	// EtherCAT device
	stText_EC_OpState_Error					: ST_Text := (
												wsNameId:= "EC_OpState_Error",
												wsName:= "EC-Error(OpState)");
	stText_EC_DeviceState_Init				: ST_Text := (
												wsNameId:= "EC_DeviceState_Init",
												wsName:= "EtherCAT Device State: INIT");
	stText_EC_DeviceState_Preop				: ST_Text := (
												wsNameId:= "EC_DeviceState_Preop",
												wsName:= "EtherCAT Device State: Pre-Operational");
	stText_EC_DeviceState_Bootstrap			: ST_Text := (
												wsNameId:= "EC_DeviceState_Bootstrap",
												wsName:= "EtherCAT Device State: Bootstrap");
	stText_EC_DeviceState_Safeop			: ST_Text := (
												wsNameId:= "EC_DeviceState_Safeop",
												wsName:= "EtherCAT Device State: Safe-Operational");
	stText_EC_DeviceState_Op				: ST_Text := (
												wsNameId:= "EC_DeviceState_Op",
												wsName:= "EtherCAT Device State: Operational");
	stText_EC_DeviceState_Error				: ST_Text := (
												wsNameId:= "EC_DeviceState_Error",
												wsName:= "EtherCAT Device State: Error");
	stText_EC_DeviceState_InvalidVprs		: ST_Text := (
												wsNameId:= "EC_DeviceState_InvalidVprs",
												wsName:= "EtherCAT Device State: Invalid VendorID, Productcode, revisionnumber or serialnumber");
	stText_EC_DeviceState_InitCmdError		: ST_Text := (
												wsNameId:= "EC_DeviceState_InitCmdError",
												wsName:= "EtherCAT Device State: INIT command error");
	stText_EC_DeviceState_Undefined			: ST_Text := (
												wsNameId:= "EC_DeviceState_Undefined",
												wsName:= "EtherCAT Device State: Undefined");
												
	// EtherCAT link state
	stText_EC_LinkState_Ok					: ST_Text := (
												wsNameId:= "EC_LinkState_Ok",
												wsName:= "EtherCAT Link State: OK");
	stText_EC_LinkState_NotPresent			: ST_Text := (
												wsNameId:= "EC_LinkState_NotPresent",
												wsName:= "EtherCAT Link State: no EtherCAT communication with slave");
	stText_EC_LinkState_WithoutCom			: ST_Text := (
												wsNameId:= "EC_LinkState_WithoutCom",
												wsName:= "EtherCAT Link State: error on port X. Port has a link, but no communication");
	stText_EC_LinkState_MissingLink			: ST_Text := (
												wsNameId:= "EC_LinkState_MissingLink",
												wsName:= "EtherCAT Link State: Missing link on port X");
	stText_EC_LinkState_AdditionalLink		: ST_Text := (
												wsNameId:= "EC_LinkState_AdditionalLink",
												wsName:= "EtherCAT Link State: Additional link on port X");
	stText_EC_LinkState_PortA				: ST_Text := (
												wsNameId:= "EC_LinkState_PortA",
												wsName:= "EtherCAT Link State: Error communication port A");
	stText_EC_LinkState_PortB				: ST_Text := (
												wsNameId:= "EC_LinkState_PortB",
												wsName:= "EtherCAT Link State: Error communication port B");
	stText_EC_LinkState_PortC				: ST_Text := (
												wsNameId:= "EC_LinkState_PortC",
												wsName:= "EtherCAT Link State: Error communication port C");
	stText_EC_LinkState_PortD				: ST_Text := (
												wsNameId:= "EC_LinkState_PortD",
												wsName:= "EtherCAT Link State: Error communication port D");
	stText_EC_LinkState_Undefined			: ST_Text := (
												wsNameId:= "EC_LinkState_Undefined",
												wsName:= "EtherCAT Link State: Undefined");

	// ProfiNet device
	stText_PN_Device_Error					: ST_Text := (
												wsNameId:= "PN_Device_Error",
												wsName:= "ProfiNet Device Status");

	// IO-Link device
	stText_IOL_Device_Error					: ST_Text := (
												wsNameId:= "IOL_Device_Error",
												wsName:= "IO-Link Device Status");
												
END_STRUCT
END_TYPE

// ---- POUs/HMI/_Structures/_Common/ST_DefaultHmiToPlc.TcDUT
TYPE ST_DefaultHmiToPlc :
STRUCT
	// default HMI items	
	bStart			: BOOL;
	bStop, bFastStop: BOOL;
	bReset			: BOOL;
	bStep			: BOOL;
	bHome			: BOOL;
	
	bOpModeManual	: BOOL;
	bOpModeAuto		: BOOL;
	bOpModeStep		: BOOL;
	
	eSafetyOpMode	: E_Opmode;
END_STRUCT
END_TYPE

// ---- POUs/Items/TcaCarrier/Enumerations/eTcaCarrierCmd.TcDUT
{attribute 'qualified_only'}
{attribute 'strict'}
{attribute 'to_string'}
TYPE eTcaCarrierCmd :
(
	noCmd := 0,
	emptyPlaces,
	fillPlaces,
	RestorePlaces,
	ConfigCarrier
);
END_TYPE

// ---- POUs/Items/TcaCarrier/Enumerations/eTcaCarrierLayout.TcDUT
{attribute 'qualified_only'}
TYPE eTcaCarrierLayout :
(
	undefined := 0,
	Layout1,
	Layout2,
	Layout3,
	Layout4,
	Layout5,
	Bulk
);
END_TYPE

// ---- POUs/Items/TcaCarrier/Structures/TcaCarrierConfig.TcDUT
TYPE TcaCarrierConfig :
STRUCT	
	/// Geometry
	Layout : eTcaCarrierLayout;		
	Dimension : ST_Coordinate;
	
	PositionsInRow : INT;			// Numbers of Positions in first Row
	RowDistance : REAL;		// Distance from one Row to the other
	PositionsInColumn : INT;			// Numbers of Positions in one Column
	ColumnDistance : REAL;		// Distance from one Column to the other
	CoordinateFirstWorkpiece : ST_Coordinate;
		
	InitialStatus : eTcaWorkpieceStatus;
	RequestStatus : eTcaWorkpieceStatus;	
	
END_STRUCT
END_TYPE

// ---- POUs/Items/TcaCarrier/Structures/TcaCarrierData.TcDUT
TYPE TcaCarrierData :
STRUCT	
	Enabled : BOOL;
	Id : INT;
	//Source		: E_Station;
	//Logging : WSTRING;	// Information in csv, xml or json Format
	Error : BOOL;	

	WorkpiecesEnabled : ARRAY[0..TcaCarrier.MAX_WORKPIECEPLACES] OF BOOL;
	WorkpiecesData : ARRAY[0..TcaCarrier.MAX_WORKPIECEPLACES] OF TcaWorkpieceData;		

END_STRUCT
END_TYPE

// ---- POUs/Items/TcaCarrier/Structures/TcaCarrierService.TcDUT
TYPE TcaCarrierService :
STRUCT

END_STRUCT
END_TYPE

// ---- POUs/Items/TcaTrolley/Structures/TcaTrolleyConfig.TcDUT
TYPE TcaTrolleyConfig : 
STRUCT	
	/// Geometry
	NumberOfCarriers : INT := 40;
	RackOrigin : ST_Coordinate;
	RackDivision : LREAL;
	CarrierDistance : LREAL;
	
	//InitialStatus : eTcaWorkpieceStatus;
	//RequestStatus : eTcaWorkpieceStatus;	
	
	CarrierConfig : TcaCarrierConfig;
	
END_STRUCT
END_TYPE

// ---- POUs/Items/TcaTrolley/Structures/TcaTrolleyData.TcDUT
TYPE TcaTrolleyData : 
STRUCT
	Exist : BOOL;
	Id : INT;
	//Logging : WSTRING;	// Information in csv, xml or json Format
	Error : BOOL;
	
	CarriersEnabled : ARRAY[0..TcaCarrier.MAX_WORKPIECEPLACES] OF BOOL;
	CarriersData : ARRAY[0..TcaTrolley.MAX_CARRIERPLACES] OF TcaCarrierData;
	
END_STRUCT
END_TYPE

// ---- POUs/Items/TcaTrolley/Structures/TcaTrolleyService.TcDUT
TYPE TcaTrolleyService :
STRUCT
	DisableCarriers		: BOOL;
	EnableCarriers		: BOOL;
	FillWithEmptyCarriers : BOOL;
	FillWithFinishedCarriers : BOOL;
	FillWithInitialCarriers : BOOL;
END_STRUCT
END_TYPE

// ---- POUs/Items/TcaWorkpiece/Enumerations/eTcaWorkpieceShape.TcDUT
{attribute 'qualified_only'}
{attribute 'strict'}
{attribute 'to_string'}
TYPE eTcaWorkpieceShape :
(
	undefined := 0,
	roll,
	ring,
	plate,
	other,
	
	MAXSIZE
);
END_TYPE

// ---- POUs/Items/TcaWorkpiece/Enumerations/eTcaWorkpieceStatus.TcDUT
{attribute 'qualified_only'}
{attribute 'to_string'}
TYPE eTcaWorkpieceStatus :
(
	undefined := 0, //leer
	noProcessDone, // grau
	laserProcessDone, // blau
	bondingAgentProcessDone, // orange
	castingProcessDone, //  violett
	finishProcessDone, //grün
	

	MAXSIZE
);
END_TYPE

// ---- POUs/Items/TcaWorkpiece/Structures/TcaWorkpieceData.TcDUT
TYPE TcaWorkpieceData : 
STRUCT
	Id : INT;	// <> 0 Workpiece Present 
	Error : BOOL;
	Exist : BOOL;
	SerialNumber : STRING;
	CurrentStatus : eTcaWorkpieceStatus;
	InitialStatus : eTcaWorkpieceStatus;
	RequestStatus : eTcaWorkpieceStatus;
	//Shape : eTcaWorkpieceShape;
	//Dimension : ST_Coordinate;
	TimeStampChanged : DT;
	Logging : WSTRING;	// Information in csv, xml or json Format
	
END_STRUCT
END_TYPE

// ---- POUs/Plant/_Enumerations/E_Module.TcDUT
//{attribute 'qualified_only'}
//{attribute 'strict'}
TYPE E_Module :
(
	eModule_none := 0,
	eModule_M001,
		
	/// has to be set to last index for array bounds!
	eModule_nMaxIdx
);
END_TYPE

// ---- POUs/Plant/_Enumerations/E_PlantSettings.TcDUT
//{attribute 'qualified_only'}
//{attribute 'strict'}
{attribute 'to_string'}
{attribute 'to_wstring'}
TYPE E_PlantSettings :
(
	//ePlant_Settings_none := 0,
	ePlantSetting_RecipeName,		// Name of the recipe
	ePlantSetting_RecipeComment,	// Comment
	ePlantSetting_PlantName,		// Plant name
	ePlantSetting_PlantNumber,		// Plant number
	
	//ePlantSetting_OvenHgPickUpDepthZ,	// Einfahrtiefe HG - Oven Z-Achse
	//
	//ePlantSetting_StorageHgSafetyDistZ,	// Sicherheitsabstand HG - Storage Z-Achse
	//
	//ePlantSetting_StorageOffsetUpY,	// HG-Offset oberhalb der Storage-Palette in Y-Richtung [mm]
	//ePlantSetting_StorageOffsetDnY, // HG-Offset unterhalb der Storage-Palette in Y-Richtung [mm]
	
	/// has to be set to last index for array bounds!
	ePlantSetting_nMaxIdx	
);
END_TYPE

// ---- POUs/Plant/_Enumerations/E_ProductionSettings.TcDUT
//{attribute 'qualified_only'}
//{attribute 'strict'}
{attribute 'to_string'}
{attribute 'to_wstring'}
TYPE E_ProductionSettings :
(
	//eProduction_Settings_none := 0,
	eProductionSettings_Override,		// override
	eProductionSettings_OrderNumber,	// order

	/// has to be set to last index for array bounds!
	eProductionSettings_nMaxIdx	
);
END_TYPE

// ---- POUs/Plant/_Enumerations/E_ProductSettings.TcDUT
//{attribute 'qualified_only'}
//{attribute 'strict'}
{attribute 'to_string'}
{attribute 'to_wstring'}
TYPE E_ProductSettings :
(
	//eProduct_Settings_none := 0,
	eProductSettings_ProductNumber,	// product nb.
	eProductSettings_ProductName,	// product name
	eProductSettings_ProductType, 	// product type
	
	//eProductSettings_Speed,			// speed [m/min]
	
	//eProductSettings_TrolleyDevisionX,	// Teilung des Trolley-Racks in X-Richtung [mm]
	//eProductSettings_TrolleyFirstPosY, 	// Erte Position im Trolley-Racks in Y-Richtung [mm]
	//eProductSettings_TrolleyCountY, 	// Letzte Position im Trolley-Racks in Y-Richtung [mm]
	//eProductSettings_TrolleyDevisionY,	// Teilung des Trolley-Racks in Y-Richtung [mm]
	//eProductSettings_TrolleyOffsetUpY,	// HG-Offset oberhalb der Trolley-Palette in Y-Richtung [mm]
	//eProductSettings_TrolleyOffsetDnY,	// HG-Offset unterhalb der Trolley-Palette in Y-Richtung [mm]
	
	eProductSettings_TrolleyNumberOfCarriers,
	eProductSettings_TrolleyRackOriginX,
	eProductSettings_TrolleyRackOriginY,
	eProductSettings_TrolleyRackOriginZ,
	eProductSettings_TrolleyRackDivision,
	eProductSettings_TrolleyCarrierDistance,
	
	eProductSettings_CarrierLayout,	
	eProductSettings_CarrierDimensionX,
	eProductSettings_CarrierDimensionY,
	eProductSettings_CarrierPositionsInRow,			// Numbers of Positions in first Row
	eProductSettings_CarrierRowDistance,		// Distance from one Row to the other
	eProductSettings_CarrierPositionsInColumn,			// Numbers of Positions in one Column
	eProductSettings_CarrierColumnDistance,		// Distance from one Column to the other
	eProductSettings_CarrierCoordinateFirstWorkpieceX,
	eProductSettings_CarrierCoordinateFirstWorkpieceY,
	eProductSettings_CarrierInitialStatus,
	eProductSettings_CarrierRequestStatus,	
	
	
	eProductSettings_HeatingPlateEnable,
	eProductSettings_HeatingPlateTemperatur,	
	
	/// has to be set to last index for array bounds!
	eProductSettings_nMaxIdx	
);
END_TYPE

// ---- POUs/Plant/_Enumerations/E_Station.TcDUT
//{attribute 'qualified_only'}
//{attribute 'strict'}
TYPE E_Station :
(
	eStation_none := 0,
	eStation_ST010_OvenA := 1,
	eStation_ST020_OvenB := 2,
	eStation_ST030_Handling := 3,
	eStation_ST040_Storage := 4,
	eStation_ST050_Mould := 5,
	
	/// has to be set to last index for array bounds!
	eStation_nMaxIdx
);
END_TYPE

// ---- POUs/Plant/M001_Module/_Enumerations/E_M001_Settings.TcDUT
//{attribute 'qualified_only'}
//{attribute 'strict'}
{attribute 'to_string'}
{attribute 'to_wstring'}
TYPE E_M001_Settings :
(
	//eSt001_Settings_none := 0,
	
	eM001_Settings_Deaktiv,		// Station deaktivieren
	eM001_Settings_Autohome,	// automatic home with start button
	
	//eM001_Settings_PalletLayout,	// Palettenlayout (1-4)
	
	/// has to be set to last index for array bounds!
	eM001_Settings_nMaxIdx	
);
END_TYPE

// ---- POUs/Plant/M001_Module/_Structures/ST_M001_HMI_IN.TcDUT
TYPE ST_M001_HMI_IN :
STRUCT
	bQuit : BOOL;
	//bJogVm : BOOL;
END_STRUCT
END_TYPE

// ---- POUs/Plant/M001_Module/_Structures/ST_M001_Interface.TcDUT
TYPE ST_M001_Interface :
STRUCT
	bRunCycle,
	bEmptyPlant : BOOL;
END_STRUCT
END_TYPE

// ---- POUs/Plant/M001_Module/_Structures/ST_M001_HMI_OUT.TcDUT
TYPE ST_M001_HMI_OUT :
STRUCT
	//fSpeed : LREAL;
END_STRUCT
END_TYPE

// ---- POUs/Plant/M001_Module/_Structures/ST_M001_IO.TcDUT
TYPE ST_M001_IO :
STRUCT
	stIn 	AT%I* : ST_M001_IO_IN;
	stOut 	AT%Q* : ST_M001_IO_OUT;
END_STRUCT
END_TYPE

// ---- POUs/Plant/M001_Module/_Structures/ST_M001_IO_IN.TcDUT
TYPE ST_M001_IO_IN :
STRUCT	
	// inputs	
	//bPwrCircBreakerOk	: BOOL;
END_STRUCT
END_TYPE

// ---- POUs/Plant/M001_Module/_Structures/ST_M001_IO_OUT.TcDUT
TYPE ST_M001_IO_OUT :
STRUCT
END_STRUCT
END_TYPE

// ---- POUs/Plant/ST010_OvenA/_Structures/ST_St010_HMI_IN.TcDUT
TYPE ST_St010_HMI_IN :
STRUCT
	bJogUp : BOOL; // Tippen Vor; DT-WH, 2FDI-NO; P10A-52SJ1
	bJogDown : BOOL; // Tippen Zurück; DT-BK, 2FDI-NO; P10A-52SJ3
	
	bJogCh1Ouside : BOOL;
	bJogCh1Inside : BOOL;
	
	bJogCh2Ouside : BOOL;
	bJogCh2Inside : BOOL;
	
	bManual : BOOL;
	bQuit : BOOL;
	
	bJog : BOOL;
	bSpeed : BOOL;
	
END_STRUCT
END_TYPE

// ---- POUs/Plant/ST010_OvenA/_Structures/ST_St010_Interface.TcDUT
TYPE ST_St010_Interface :
STRUCT
	bEnableSequence,	// enable to main module
	
	bResponseChkIndex,
	bResponseIsEmptySlot,
	bResponseOpn	: BOOL;	// handshake response segment open
	iConfirmPosition	: INT;	// handshake confirm segment open @ x,y index
	
	Trolley			: TcaTrolley;
END_STRUCT
END_TYPE

// ---- POUs/Plant/ST010_OvenA/_Structures/ST_St010_HMI_IN_OUT.TcDUT
TYPE ST_St010_HMI_IN_OUT : //EXTENDS ST_HMI_TR_CMD :
STRUCT
END_STRUCT
END_TYPE

// ---- POUs/Plant/ST020_OvenB/_Enumerations/E_St020_Settings.TcDUT
//{attribute 'qualified_only'}
//{attribute 'strict'}
{attribute 'to_string'}
{attribute 'to_wstring'}
TYPE E_St020_Settings :
(
	//eSt020_Settings_none := 0,
	
	eSt020_Settings_Station_Deaktiv,	// Station deaktivieren
	eSt020_Settings_Autohome,			// automatic home with start button
	
	eSt020_Settings_HomeSpeed,			// Homing-Geschwindigkeit [mm/s]
	eSt020_Settings_JogSpeed,			// Tippgeschwindigkeit [mm/s]
	eSt020_Settings_WorkSpeed,			// Automatik-Geschwindigkeit [mm/s]
	eSt020_Settings_JogSpeedCh,			// Tippgeschwindigkeit CH-Achsen [mm/s]
	eSt020_Settings_WorkSpeedCh,		// Automatik-Geschwindigkeit CH-Achsen [mm/s]

	eSt020_Settings_AxisRefPos,			// Referenzposition Achse [mm]
	eSt020_Settings_PosHome,			// Homeposition [mm]
	eSt020_Settings_PosWork,			// Mitnehmerposition unteres Segment [mm]
	
	eSt020_Settings_PosHomeCh,			// Homeposition CH-Achsen [mm]
	eSt020_Settings_PosWorkCh,			// Arbeitsposition CH-Achsen [mm]
	
	eSt020_Settings_OvenFixPartHeight,	// Festteilhöhe [mm]
	eSt020_Settings_OvenSegmentHeight,	// Festteilhöhe [mm]
	
	eSt020_Settings_OvenMiddlePointX,	// Mittelpunnkt in X-Richtung [mm]
	eSt020_Settings_OvenOffsetY,		// Y-Offset Ofen [mm]
	eSt020_Settings_OvenPickUpDepthZ,	// Teach-Position, Storage 2 Z [mm]
	
	eSt020_Settings_XPosRp1,			// Teach-Position, Ofen B, RP 1 X [mm]
	eSt020_Settings_YPosRp1,			// Teach-Position, Ofen B, RP 1 Y [mm]
	eSt020_Settings_ZPosRp1,			// Teach-Position, Ofen B, RP 1 Z [mm]
	                                                           
	eSt020_Settings_XPosRp2,			// Teach-Position, Ofen B, RP 2 X [mm]
	eSt020_Settings_YPosRp2,			// Teach-Position, Ofen B, RP 2 Y [mm]
	eSt020_Settings_ZPosRp2,			// Teach-Position, Ofen B, RP 2 Z [mm]
	
	/// has to be set to last index for array bounds!
	eSt020_Settings_nMaxIdx	
);
END_TYPE

// ---- POUs/Plant/ST020_OvenB/_Structures/ST_St020_HMI_IN_OUT.TcDUT
TYPE ST_St020_HMI_IN_OUT : // EXTENDS ST_HMI_TR_CMD :
STRUCT
END_STRUCT
END_TYPE

// ---- POUs/Plant/ST020_OvenB/_Structures/ST_St020_HMI_IN.TcDUT
TYPE ST_St020_HMI_IN :
STRUCT	
	bJogUp : BOOL; // Tippen Vor; DT-WH, 2FDI-NO; P10A-52SJ1
	bJogDown : BOOL; // Tippen Zurück; DT-BK, 2FDI-NO; P10A-52SJ3
	
	bJogCh1Ouside : BOOL;
	bJogCh1Inside : BOOL;
	
	bJogCh2Ouside : BOOL;
	bJogCh2Inside : BOOL;
	
	bManual : BOOL;
	bQuit : BOOL;
	
	bJog : BOOL;
	bSpeed : BOOL;
END_STRUCT
END_TYPE

// ---- POUs/Plant/ST020_OvenB/_Structures/ST_St020_Interface.TcDUT
TYPE ST_St020_Interface :
STRUCT
	bEnableSequence,	// enable to main module
	
	bResponseChkIndex,
	bResponseIsEmptySlot,
	bResponseOpn	: BOOL;	// handshake response segment open
	iConfirmPosition	: INT;	// handshake confirm segment open @ x,y index
	
	Trolley			: TcaTrolley;
END_STRUCT
END_TYPE

// ---- POUs/Plant/ST020_OvenB/_Structures/ST_St020_IO.TcDUT
TYPE ST_St020_IO :
STRUCT
	stIn	AT%I* : ST_St020_IO_IN;
	stOut	AT%Q* : ST_St020_IO_OUT;
	stHeatingPlateIO : ST_FurnaceIO;
END_STRUCT
END_TYPE

// ---- POUs/Plant/ST020_OvenB/_Structures/ST_St020_IO_IN.TcDUT
TYPE ST_St020_IO_IN :
STRUCT	
	// inputs
	bRefpos	: BOOL;	// Sensor | Oven | Referenzposition | BMK: =P260+xyz- | Terminal: .: | Tc3Hmi
END_STRUCT
END_TYPE

// ---- POUs/Plant/ST020_OvenB/_Structures/ST_St020_IO_OUT.TcDUT
TYPE ST_St020_IO_OUT :
STRUCT
	bOvenFan :BOOL;
END_STRUCT
END_TYPE

// ---- POUs/Plant/ST020_OvenB/_Structures/ST_St020_HMI_OUT.TcDUT
TYPE ST_St020_HMI_OUT :
STRUCT
	//Trolley	: ST_Trolley;
END_STRUCT
END_TYPE

// ---- POUs/Plant/ST030_Handling/_Enumerations/E_St030_Command.TcDUT
{attribute 'qualified_only'}
{attribute 'strict'}
{attribute 'to_string'}
TYPE E_St030_Command :
(
	eSt030_Command_none := 0,
	eSt030_Command_OvenA_Get,
	eSt030_Command_OvenA_Put,
	
	eSt030_Command_OvenB_Get,
	eSt030_Command_OvenB_Put,
	
	eSt030_Command_Storage_Get,
	eSt030_Command_Storage_Put
);
END_TYPE

// ---- POUs/Plant/ST030_Handling/_Enumerations/E_St030_EmptySlotChk.TcDUT
{attribute 'qualified_only'}
{attribute 'strict'}
{attribute 'to_string'}
TYPE E_St030_EmptySlotChk :
(
	eSt030_EmptySlotChk_none := 0,
	eSt030_EmptySlotChk_Empty,
	eSt030_EmptySlotChk_NotEmpty
);
END_TYPE

// ---- POUs/Plant/ST030_Handling/_Enumerations/E_St030_Settings.TcDUT
//{attribute 'qualified_only'}
//{attribute 'strict'}
{attribute 'to_string'}
{attribute 'to_wstring'}
TYPE E_St030_Settings :
(
	//eSt030_Settings_none := 0,
	
	eSt030_Settings_Station_Deaktiv,	// Station deaktivieren
	eSt030_Settings_Autohome,			// automatic home with start button
	
	eSt030_Settings_XHomeSpeed,			// Homing-Geschwindigkeit X [mm/s]
	eSt030_Settings_XJogSpeed,			// Tippgeschwindigkeit X [mm/s]
	eSt030_Settings_XWorkSpeed,			// Automatik-Geschwindigkeit X [mm/s]
	
	eSt030_Settings_YHomeSpeed,			// Homing-Geschwindigkeit Y [mm/s]
	eSt030_Settings_YJogSpeed,			// Tippgeschwindigkeit Y [mm/s]
	eSt030_Settings_YWorkSpeed,			// Automatik-Geschwindigkeit Y [mm/s]
	
	eSt030_Settings_ZHomeSpeed,			// Homing-Geschwindigkeit Z [mm/s]
	eSt030_Settings_ZJogSpeed,			// Tippgeschwindigkeit Z [mm/s]
	eSt030_Settings_ZWorkSpeed,			// Automatik-Geschwindigkeit Z [mm/s]
	
	eSt030_Settings_AxisRefPosX,		// reference pos axis HG X
	eSt030_Settings_AxisRefPosY,		// reference pos axis HG Y
	eSt030_Settings_AxisRefPosZ,		// reference pos axis HG Z
	
	eSt030_Settings_XPosHome,			// Homeposition X [mm]
	eSt030_Settings_YPosHome,			// Homeposition Y [mm]
	eSt030_Settings_ZPosHome,			// Homeposition Z [mm]

	
	eSt030_Settings_XPosOv2Rp1,			// Teach-Position, Ofen 2, RP 1 X [mm]
	eSt030_Settings_YPosOv2Rp1,			// Teach-Position, Ofen 2, RP 1 Y [mm]
	eSt030_Settings_ZPosOv2Rp1,			// Teach-Position, Ofen 2, RP 1 Z [mm]

	eSt030_Settings_XPosOv2Rp2,			// Teach-Position, Ofen 2, RP 2 X [mm]
	eSt030_Settings_YPosOv2Rp2,			// Teach-Position, Ofen 2, RP 2 Y [mm]
	eSt030_Settings_ZPosOv2Rp2,			// Teach-Position, Ofen 2, RP 2 Z [mm]
	
	
	/// has to be set to last index for array bounds!
	eSt030_Settings_nMaxIdx
);
END_TYPE

// ---- POUs/Plant/ST030_Handling/_Structures/ST_St030_HMI_OUT.TcDUT
TYPE ST_St030_HMI_OUT :
STRUCT
	//Pallet	: ST_Pallet;
END_STRUCT
END_TYPE

// ---- POUs/Plant/ST030_Handling/_Structures/ST_St030_HMI_IN.TcDUT
TYPE ST_St030_HMI_IN :
STRUCT
	bJogXP		: BOOL; // Tippen Vor; DT-WH, 2FDI-NO; P10A-52SJ1
	bJogXN		: BOOL; // Tippen Zurück; DT-BK, 2FDI-NO; P10A-52SJ3
	
	bJogYP		: BOOL; // Tippen Vor; DT-WH, 2FDI-NO; P10A-52SJ1
	bJogYN		: BOOL; // Tippen Zurück; DT-BK, 2FDI-NO; P10A-52SJ3
	
	bJogZP		: BOOL; 
	bJogZN		: BOOL; 
	
	bManual : BOOL;
	bQuit :  BOOL;
		
	bJog : BOOL;
	bSpeed : BOOL;
END_STRUCT
END_TYPE

// ---- POUs/Plant/ST030_Handling/_Structures/ST_St030_Interface.TcDUT
TYPE ST_St030_Interface :
STRUCT
	bEnable,
	bEnableOvenAxis,

	bReqestOvenA,			// request entry to stations
	bReqestOvenA_ChkIndex,
	bReqestOvenB,
	bReqestOvenB_ChkIndex,
	bReqestStorage,
	bReqestStorage_ChkIndex	: BOOL;	
	
	// current pallet on GH
	Pallet			: TcaCarrier;
	Source			: E_Station;
	
	// active / requested HG command
	CommandRequest	: ST_St030_Command;
	ActiveCommand	: ST_St030_Command;
END_STRUCT
END_TYPE

// ---- POUs/Plant/ST030_Handling/_Structures/ST_St030_Command.TcDUT
TYPE ST_St030_Command :
STRUCT
	Command : E_St030_Command;
	Position : INT;
	//IndexX,
	//IndexY	: INT;
END_STRUCT
END_TYPE

// ---- POUs/Plant/ST030_Handling/_Structures/ST_St030_IO.TcDUT
TYPE ST_St030_IO :
STRUCT
	stIn	AT%I* : ST_St030_IO_IN;
	stOut	AT%Q* : ST_St030_IO_OUT;
END_STRUCT
END_TYPE

// ---- POUs/Plant/ST030_Handling/_Structures/ST_St030_IO_IN.TcDUT
TYPE ST_St030_IO_IN :
STRUCT
	// inputs handling
	bRefposX	: BOOL;	// Sensor | Handling | Referenzposition X | BMK: =P260+xyz- | Terminal: .: | Tc3Hmi
	bRefposY	: BOOL;	// Sensor | Handling | Referenzposition Y | BMK: =P260+xyz- | Terminal: .: | Tc3Hmi
	bRefposZ	: BOOL;	// Sensor | Handling | Referenzposition Z | BMK: =P260+xyz- | Terminal: .: | Tc3Hmi
	
	fMeasurementA : DINT;	// Sensor | Handling | S1 | BMK: =P260+xyz- | Terminal: .: | Tc3Hmi
	fMeasurementB : DINT;	// Sensor | Handling | S2 | BMK: =P260+xyz- | Terminal: .: | Tc3Hmi
END_STRUCT
END_TYPE

// ---- POUs/Plant/ST030_Handling/_Structures/ST_St030_IO_OUT.TcDUT
TYPE ST_St030_IO_OUT :
STRUCT
	// outputs handling
END_STRUCT
END_TYPE

// ---- POUs/Plant/ST030_Handling/_Structures/ST_St030_HMI_IN_OUT.TcDUT
TYPE ST_St030_HMI_IN_OUT ://EXTENDS ST_HMI_PL_CMD :
STRUCT
END_STRUCT
END_TYPE

// ---- POUs/Plant/ST030_Handling/_Structures/ST_XZ_Point.TcDUT
TYPE ST_XZ_Point :
STRUCT
	X,
	Z : LREAL;
END_STRUCT
END_TYPE

// ---- POUs/Plant/ST040_Storage/_Enumerations/E_St040_Settings.TcDUT
//{attribute 'qualified_only'}
//{attribute 'strict'}
{attribute 'to_string'}
{attribute 'to_wstring'}
TYPE E_St040_Settings :
(
	//eSt040_Settings_none := 0,
	
	eSt040_Settings_Station_Deaktiv,	// Station deaktivieren
	eSt040_Settings_Autohome,			// automatic home with start button
	
	eSt040_Settings_JogSpeed,			// Tippgeschwindigkeit [mm/s]
	eSt040_Settings_WorkSpeed,			// Automatik-Geschwindigkeit  [mm/s]
	
	eSt040_Settings_PosHome,			// Homeposition [mm]
	eSt040_Settings_PosWork,			// Arbeitsposition [mm]
	
	eSt040_Settings_XPosStor1,			// Teach-Position, Storage 1 X [mm]
	eSt040_Settings_YPosStor1,			// Teach-Position, Storage 1 Y [mm]
	eSt040_Settings_ZPosStor1,			// Teach-Position, Storage 1 Z [mm]
	    
	eSt040_Settings_XPosStor2,			// Teach-Position, Storage 2 X [mm]
	eSt040_Settings_YPosStor2,			// Teach-Position, Storage 2 Y [mm]
	eSt040_Settings_ZPosStor2,			// Teach-Position, Storage 2 Z [mm]
	
	
	/// has to be set to last index for array bounds!
	eSt040_Settings_nMaxIdx	
);
END_TYPE

// ---- POUs/Plant/ST040_Storage/_Structures/ST_St040_HMI_IN.TcDUT
TYPE ST_St040_HMI_IN :
STRUCT
	bJog01Up		: BOOL; // Tippen Vor; DT-WH, 2FDI-NO; P10A-52SJ1
	bJog01Down		: BOOL; // Tippen Zurück; DT-BK, 2FDI-NO; P10A-52SJ3
	
	bJog02Up	 	: BOOL; 
	bJog02Down	: BOOL; 	
	
	bManual : BOOL;
	bQuit :  BOOL;
	
	bJog : BOOL;
	bSpeed : BOOL;

END_STRUCT
END_TYPE

// ---- POUs/Plant/ST040_Storage/_Structures/ST_St040_HMI_IN_OUT.TcDUT
TYPE ST_St040_HMI_IN_OUT : //EXTENDS ST_HMI_PL_CMD :
STRUCT
	// pallet index on storage
	Idx		: INT;
END_STRUCT
END_TYPE

// ---- POUs/Plant/ST040_Storage/_Structures/ST_St040_HMI_OUT.TcDUT
TYPE ST_St040_HMI_OUT :
STRUCT
	//Pallet1,
	//Pallet2	: ST_Pallet;
END_STRUCT
END_TYPE

// ---- POUs/Plant/ST040_Storage/_Structures/ST_St040_IO.TcDUT
TYPE ST_St040_IO :
STRUCT
	stIn	AT%I* : ST_St040_IO_IN;
	stOut	AT%Q* : ST_St040_IO_OUT;
END_STRUCT
END_TYPE

// ---- POUs/Plant/ST040_Storage/_Structures/ST_St040_IO_IN.TcDUT
TYPE ST_St040_IO_IN :
STRUCT
END_STRUCT
END_TYPE

// ---- POUs/Plant/ST040_Storage/_Structures/ST_St040_IO_OUT.TcDUT
TYPE ST_St040_IO_OUT :
STRUCT
	// outputs OptischeKontrolle	
	nCamPrgAs	: INT;
	nCamPrgBs	: INT;
	
	bLedAs		: BOOL;
	bLedBs		: BOOL;
END_STRUCT
END_TYPE

// ---- POUs/Plant/ST040_Storage/_Structures/ST_St040_Interface.TcDUT
TYPE ST_St040_Interface :
STRUCT
	bEnable,				// enable to main module
	
	bResponseChkIndex,
	bResponseEmptyAtIndex,
	bResponseOpn	: BOOL;	// handshake response open
	iConfirmPosition 	: INT;	// handshake confirm open @ index
	
	Pallet1,
	Pallet2	: TcaCarrier;
	
	Source1,	
	Source2			: E_Station;
END_STRUCT
END_TYPE

// ---- POUs/Plant/ST050_Mould/_Enumerations/E_St050_Settings.TcDUT
//{attribute 'qualified_only'}
//{attribute 'strict'}
{attribute 'to_string'}
{attribute 'to_wstring'}
TYPE E_St050_Settings :
(
	//eSt050_Settings_none := 0,
	
	eSt050_Settings_Station_Deaktiv,	// Station deaktivieren
	eSt050_Settings_Autohome,			// automatic home with start button

	
	/// has to be set to last index for array bounds!
	eSt050_Settings_nMaxIdx	
);
END_TYPE

// ---- POUs/Plant/ST050_Mould/_Structures/ST_St050_Interface.TcDUT
TYPE ST_St050_Interface :
STRUCT
	bEnableHG	: BOOL; // enable handling
	
	bReqS1Empty,
	bReqS2Empty,
	bReqS1Unfinished,
	bReqS2Unfinished,
	bReqS1NoCarrier,
	bReqS2NoCarrier	: BOOL;
END_STRUCT
END_TYPE

// ---- POUs/Plant/ST050_Mould/_Structures/ST_St050_IO.TcDUT
TYPE ST_St050_IO :
STRUCT
	stIn	AT%I* : ST_St050_IO_IN;
	stOut	AT%Q* : ST_St050_IO_OUT;
END_STRUCT
END_TYPE

// ---- POUs/Plant/ST050_Mould/_Structures/ST_St050_IO_IN.TcDUT
TYPE ST_St050_IO_IN :
STRUCT
	aFromEngelRaw	: ARRAY[0..41] OF BYTE;
	bRequestOpenProtectionDoor : BOOL;
END_STRUCT
END_TYPE

// ---- POUs/Plant/ST050_Mould/_Structures/ST_St050_IO_OUT.TcDUT
TYPE ST_St050_IO_OUT :
STRUCT
	aToEngelRaw	: ARRAY[0..41] OF BYTE;
	bReleaseSafetyGate : BOOL;
END_STRUCT
END_TYPE

// ---- POUs/Plant/ST050_Mould/_Structures/TcaEngelCastingCarrierInput.TcDUT
TYPE TcaEngelCastingCarrierInput : // ENGEL SPS -> ASMA SPS
STRUCT
	LifeCounter : UINT;
	
	
	// Modus bzw Status der Gießmaschine und Roboter
	AutoMode : BOOL;		// Roboter und Gießmaschine im zyklischen Automatikbetrieb
	SemiAutoMode : BOOL;	// Roboter und Gießmaschine im sequentiellen Halb-Automatikbetrieb
	ManualMode : BOOL;		// Roboter und Gießmaschine befinden sich in Handbetrieb
	Error : BOOL;			// Roboter bzw. Gießmaschine hat Error
	ErrorID : UINT;			// ErrorID
	
	// Überwachung und Kontrolle der Roboterposition
	Moving : BOOL;				// Roboter in Bewegung
	ParkPosition : BOOL;		// Roboter in Wartepostion
	OutsideStorage_1 : BOOL;	// Roboter außerhalb Ablage 1
	OutsideStorage_2 : BOOL;	// Roboter außerhalb Ablage 2

	// Allgemeine Sicherheit                    	
	SafetyAreaSafe : BOOL;	// Schutztüren geschlossen & quittiert		

	// Anforderung eines Werkstückträgers
	// Wird ein leerer Werkstückablageplatz oder ein Einleigeteil benötigt muss für den jeweiligen Ablageplatz
	// ein Job angefrgt werden.
	// Wenn kein Werkstückträger benötigt wird, kann auch dieser Job erteilt werden (z.B. bei Produktionsende)
	
	JobForStorage_1 : TcaEngelCastingCarrierJob;	// Anforderung eines Werkstückträgers für Ablage 1
	JobForStorage_2 : TcaEngelCastingCarrierJob;	// Anforderung eines Werkstückträgers für Ablage 2
	
	// Status des Werkstückträgers
	// Beim Entnehmen und Bestücken eines Werkstückes durch den Engel Roboter wird die Statusstruktur aktualisiert
	
	Storage_1 : TcaEngelCastingCarrierStatus;	// aktueller Status des Werkstückträgers in Ablage 1
	Storage_2 : TcaEngelCastingCarrierStatus;	// aktueller Status des Werkstückträgers in Ablage 2
	
END_STRUCT
END_TYPE

// ---- POUs/Plant/ST050_Mould/_Structures/TcaEngelCastingCarrierJob.TcDUT
TYPE TcaEngelCastingCarrierJob :
STRUCT
	RequestNoCarrier : BOOL;	// TRUE wenn kein neuer Werkstückträger benötigt wird -> Ablage wird leer gemacht
	RequestCarrier : BOOL;		// TRUE wenn ein neuer Werkstückträger benötigt wird
	CarrierId : INT;			// ID vom Werkstückträger, Geometrischen Daten werden auf der Engel Steuerung verwaltet
	Empty : BOOL;				// TRUE wenn ein Werkstückträger mir leeren Plätzen benötigt wird
	Unfinished : BOOL;			// TRUE wenn ein Werkstückträger mit unfertigen Werkstücken benötigt wird
END_STRUCT
END_TYPE

// ---- POUs/Plant/ST050_Mould/_Structures/TcaEngelCastingCarrierJobStatus.TcDUT
TYPE TcaEngelCastingCarrierJobStatus :
STRUCT
	CarrierPresent : BOOL;						// TRUE wenn ein Werkstückträger abgelegt wurde
	Carrier : TcaEngelCastingCarrierStatus;		// Status des Carriers der abgelegt wurde
	Done : BOOL;								// Job wurde erfolgreich ausgeführt
	Busy : BOOL;								// Job wird ausgeführt
	Error : BOOL;								// Job endet mit Fehler
	ErrorID : UINT;								// TODO: Welche unterschiedlichen Fehler sollen berücksichtigt werden? z.b: kein Blech, Ofentür offen, Wagen ist zum wechseln, ...								
END_STRUCT
END_TYPE

// ---- POUs/Plant/ST050_Mould/_Structures/TcaEngelCastingCarrierOutput.TcDUT
TYPE TcaEngelCastingCarrierOutput :	// ASMA SPS -> ENGEL SPS
STRUCT
	LifeCounter : UINT;
	
	// Status der Peripherie
	Ready : BOOL;			// Bereit zum Entgegennehmen von Jobs
	Busy : BOOL;			// Peripherie ist in Arbeit/ Bewegung
	Error : BOOL;			// Peripherie hat Error
	ErrorID : INT;			// ErrorID
	
	// Überwachung und Kontrolle der Ablageposition und des Handlings
	PermitRoboterHandling : BOOL; 	// Bewegungen des Engel Roboters erlauben (freie Fahrt im gesamten Bewgungsbereich)(
	PermitStorage_1 : BOOL;			// Zugriff auf Ablage 1 erlauben (aufnehmen und ablegen)
	PermitStorage_2 : BOOL;			// Zugriff auf Ablage 1 erlauben (aufnehmen und ablegen)
	                    	
	// Allgemeine Sicherheit						
	SafetyAreaRequest : BOOL; 	// Anforderung Schutztüre
	SafetyDoorRelease : BOOL;	// freigabe zum öffnen der Schutztüre
	
	// Status der Jobs
	JobStatusForStorage_1 : TcaEngelCastingCarrierJobStatus;	// Status des Jobs für Ablage 1
	JobStatusForStorage_2 : TcaEngelCastingCarrierJobStatus;	// Status des Jobs für Ablage 2
END_STRUCT
END_TYPE

// ---- POUs/Plant/ST050_Mould/_Structures/TcaEngelCastingCarrierStatus.TcDUT
TYPE TcaEngelCastingCarrierStatus :
STRUCT
	CarrierId : UINT ; // ID vom Werkstückträger, Geometrischen Daten werden auf der Engel Steuerung verwaltet
	CountMax : UINT ; // maximale Anzahl an Werkstücken die am Werkstückträger abgelegt werden können
	CountUnfinished : UINT ; // Anzahl der nicht gegossenen Rohlinge am Werkstückträger
	CountFinished : UINT ; // Anzahl der fertigen Werkstücke am Werkstückträger
	CountEmpty : UINT ; // Anzahl der leeren Plätze am Werkstückträger
END_STRUCT
END_TYPE

// ---- POUs/Plant/_Structures/ControlCabinet/ST_ControlCabinetIn.TcDUT
TYPE ST_ControlCabinetIn :
STRUCT
	/// EtherCAT master AMS Netid
	stEtherCATMasterAmsAdr 			: ST_AmsAddr;
	/// EtherCAT master device state
	eEtherCATDeviceState			: E_EcDeviceState;
	/// EtherCAT master device id
	uiEcMasterDevId					: UINT;
	/// EtherCAT Box Status & control cabinet IOs
	IarrEcStates					: ARRAY[0..E_EtherCatBox.eEtherCatBox_nMaxIdx] OF UINT;

	// =A01.K20
	//stA01	: ST_ControlCabinet_A01_In;

END_STRUCT
END_TYPE

// ---- POUs/Plant/_Structures/ControlCabinet/ST_ControlCabinetIO.TcDUT
/// Control cabinet IOs
TYPE ST_ControlCabinetIO :
STRUCT
	stIn	AT%I* : ST_ControlCabinetIn;
	stOut	AT%Q* : ST_ControlCabinetOut;
END_STRUCT
END_TYPE

// ---- POUs/Plant/_Structures/ControlCabinet/ST_ControlCabinetOut.TcDUT
TYPE ST_ControlCabinetOut :
STRUCT
	// bLed_AmpelBlau    :BOOL;(*Led | Ampelsaeule | Blau | BMK: =P238+A1+E1-17U3 | Terminal: .: | Tc3Hmi *) 
	// bLed_AmpelGruen    :BOOL;(*Led | Ampelsaeule | Gruen | BMK: =P238+A1+E1-17U3 | Terminal: .: | Tc3Hmi *) 
	// bLed_AmpelGelb    :BOOL;(*Led | Ampelsaeule | Gelb | BMK: =P238+A1+E1-17U3 | Terminal: .: | Tc3Hmi *) 
	// bLed_AmpelRot    :BOOL;(*Led | Ampelsaeule | Rot | BMK: =P238+A1+E1-17U3 | Terminal: .: | Tc3Hmi *) 

	// =A01.K20
	//stA01 : ST_ControlCabinet_A01_Out;
END_STRUCT
END_TYPE

// ---- POUs/Plant/_Structures/Counter/ST_Counter.TcDUT
TYPE ST_Counter :
STRUCT
	//Counter Overall/Shift
	diOverallCounterOk	: UDINT;
	diOverallCounterNok	: UDINT;
END_STRUCT
END_TYPE

// ---- POUs/Plant/_Structures/Objects/ST_Objects.TcDUT
TYPE ST_Objects :
STRUCT	
	stPlant_Objects		: ARRAY[0..iMaxIdxObject] OF ST_Object_Item; // e.g.: P001_Plant
	stModule_Objects	: ARRAY[0..iMaxIdxObject] OF ST_Object_Item; // e.g.: M001_Prepare
	//ToDo: clean up objects --> stStation_Objects	: ARRAY[0..E_Station.eStation_nMaxIdx] OF ST_Objects_Station; // e.g.: ST001_Separation, ...
END_STRUCT
END_TYPE

// ---- POUs/Plant/_Structures/Objects/ST_Object_Item.TcDUT
TYPE ST_Object_Item :
STRUCT
	nIndexColor		: UDINT;	//ToDo: nIndexColor not used in HMI!!!
	stGroup			: ST_Text;	//example -> station 001
	stType			: ST_Text;	//example -> axis
	stName			: ST_Text;	//example -> axis x
	stState			: ST_Text;	//example -> drive positiv
	stValue			: ST_Text;	//example -> 105.66 mm
	diObjectIndex	: DINT;		//example -> 10005
END_STRUCT
END_TYPE

// ---- POUs/Plant/_Structures/Settings/ST_ModuleDynSettings.TcDUT
TYPE ST_ModuleDynSettings :
STRUCT

	// module settings
	stDynStationSettings	: ARRAY[0..CONST.iMaxIdxLocalSetting] OF ST_Data_Item;

END_STRUCT
END_TYPE

// ---- POUs/Plant/_Structures/Settings/ST_Settings.TcDUT
TYPE ST_Settings :
STRUCT
	// plant/product/production settings
	stPlant_Settings		: ARRAY[0..E_PlantSettings.ePlantSetting_nMaxIdx] OF ST_Data_Item;			// plant
	stProduct_Settings		: ARRAY[0..E_ProductSettings.eProductSettings_nMaxIdx] OF ST_Data_Item;		// product data
	stProduction_Settings	: ARRAY[0..E_ProductionSettings.eProductionSettings_nMaxIdx] OF ST_Data_Item;	// production data

	// module & station settings
	stModuleSettings		: ARRAY[0..E_Module.eModule_nMaxIdx] OF ST_ModuleDynSettings;
	stStationSettings		: ARRAY[0..E_Station.eStation_nMaxIdx] OF ST_StationDynSettings;
	
	stCarrier				: TcaCarrierConfig;
	stTrolley				: TcaTrolleyConfig;
	
	// special settings
	//PalletLayoutIndexEnable	: ARRAY[0..CONST.iMaxIdxPalletWorkpieceX, 0..CONST.iMaxIdxPalletWorkpieceY] OF BOOL;
END_STRUCT
END_TYPE

// ---- POUs/Plant/_Structures/Settings/ST_StationDynSettings.TcDUT
TYPE ST_StationDynSettings :
STRUCT

	// station settings
	stDynStationSettings	: ARRAY[0..CONST.iMaxIdxLocalSetting] OF ST_Data_Item;

END_STRUCT
END_TYPE

// ---- POUs/Plant/_Structures/ST_DefaultEventClasses.TcDUT
TYPE ST_DefaultEventClasses :
STRUCT
	Info,
	Warning,
	Error : TcEventEntry;
END_STRUCT
END_TYPE

// ---- POUs/Safety/Components/Euchner_MBM/Structure/ST_Euchner_MBM_HW_IN.TcDUT
TYPE ST_Euchner_MBM_HW_IN :
STRUCT
	///Hardware In
	nByte0: USINT;
END_STRUCT
END_TYPE

// ---- POUs/Safety/Components/Euchner_MBM/Structure/ST_Euchner_MBM_HW_OUT.TcDUT
TYPE ST_Euchner_MBM_HW_OUT :
STRUCT
	///Hardware Out
	nByte0: USINT;
END_STRUCT
END_TYPE

// ---- POUs/Safety/Components/Euchner_MBM/Structure/ST_Euchner_MBM_IN.TcDUT
TYPE ST_Euchner_MBM_IN :
STRUCT
	///BM_D_RUN | Diagnose Runmode
	bBM_D_RUN: BOOL;
	///BM_E_ML1 | Fehlermeldebit Strang 1
	bBM_E_ML1: BOOL;
	///BM_E_ML2 | Fehlermeldebit Strang 2
	bBM_E_ML2: BOOL;
	///BM_E_SYS | Fehlermeldebit Gesamtsystem
	bBM_E_SYS: BOOL;
	///Fehlermeldebit allgemeiner Modulfehler
	bBM_E_G: BOOL;
END_STRUCT
END_TYPE

// ---- POUs/Safety/Components/Euchner_MBM/Structure/ST_Euchner_MBM_OUT.TcDUT
TYPE ST_Euchner_MBM_OUT :
STRUCT
	///Quittierbit für Fehler allgemein
	bBM_ACK_G: BOOL;
END_STRUCT
END_TYPE

// ---- POUs/Safety/Components/Euchner_MBM/Structure/ST_MBM_IO.TcDUT
TYPE ST_MBM_IO :
STRUCT
	stHwInMbm		AT%I*	: ST_Euchner_MBM_HW_IN;
	stHwOutMbm		AT%Q*	: ST_Euchner_MBM_HW_OUT;
END_STRUCT
END_TYPE

// ---- POUs/Safety/Components/Euchner_MGB2/Structure/MGB2/ST_Euchner_MGB2_HW_IN.TcDUT
TYPE ST_Euchner_MGB2_HW_IN :
STRUCT
	///Hardware In
	nByte0: USINT;
	///Hardware In
	nByte1: USINT;
END_STRUCT
END_TYPE

// ---- POUs/Safety/Components/Euchner_MGB2/Structure/MGB2/ST_Euchner_MGB2_HW_OUT.TcDUT
TYPE ST_Euchner_MGB2_HW_OUT :
STRUCT
	///Hardware Out
	nByte0: USINT;
END_STRUCT
END_TYPE

// ---- POUs/Safety/Components/Euchner_MGB2/Structure/MGB2/ST_Euchner_MGB2_IN.TcDUT
TYPE ST_Euchner_MGB2_IN :
STRUCT
	///LM_D_RUN | Diagnose Runmode
	bLM_D_RUN: BOOL;
	///LM_I_SK | nicht sicherer Eingang Tür- und Riegelstellung
	bLM_I_SK: BOOL;
	///LM_I_UK | nicht sicherer Eingang Zuhaltungsüberwachung
	bLM_I_UK: BOOL;
	///LM_E_SM1 | Fehlermeldebit für Submodul 1
	bLM_E_SM1: BOOL;
	///LM_E_SM1 | Fehlermeldebit für Submodul 1
	bLM_E_SM2: BOOL;
	///LM_E_ER | Fehlermeldebit für Fluchtentriegelung
	bLM_E_ER: BOOL;
	///LM_E_G | Fehlermeldebit allgemeiner Modulfehler
	bLM_E_G: BOOL;
	///LM_I_OD | nicht sicherer Eingang Türstellung
	bLM_I_OD: BOOL;
	///LM_I_OT | nicht sicherer Eingang Riegelzunge
	bLM_I_OT: BOOL;
	///LM_I_OL | nicht sicherer Eingang Zuhaltung
	bLM_I_OL: BOOL;
END_STRUCT
END_TYPE

// ---- POUs/Safety/Components/Euchner_MGB2/Structure/MGB2/ST_Euchner_MGB2_OUT.TcDUT
TYPE ST_Euchner_MGB2_OUT :
STRUCT
	///LM_O_CL | nicht sichere Ansteuerung der Zuhaltung
	bLM_O_CL: BOOL;
	///LM_ACK_ER | Quittierbit für Fehler Fluchtentriegelung
	bLM_ACK_ER: BOOL;
	///LM_ACK_G | Quittierbit für Fehler allgemein
	bLM_ACK_G: BOOL;
END_STRUCT
END_TYPE

// ---- POUs/Safety/Components/Euchner_MGB2/Structure/MSM/ST_Euchner_MSM_DA_IN.TcDUT
TYPE ST_Euchner_MSM_DA_IN :
STRUCT
	///SM_I_X3 | Eingang Zustimmtaster
	bSM_I_X3: BOOL;
	///SM_I_T2 | Eingang Taster
	bSM_I_T2: BOOL;
	///SM_I_T1 | Eingang Taster
	bSM_I_T1: BOOL;
	///SM_E_X3 | Fehler Zustimmtaster
	bSM_E_X3: BOOL;
END_STRUCT
END_TYPE

// ---- POUs/Safety/Components/Euchner_MGB2/Structure/MSM/ST_Euchner_MSM_DA_OUT.TcDUT
TYPE ST_Euchner_MSM_DA_OUT :
STRUCT
	///SM_O_L2 | Led 2
	bSM_O_L2: BOOL;
	///SM_O_L1 | Led 1
	bSM_O_L1: BOOL;
	///SM_O_L2_B | Led 2 blink
	bSM_O_L2_B: BOOL;
	///SM_O_L1_B | Led 1 blink
	bSM_O_L1_B: BOOL;
END_STRUCT
END_TYPE

// ---- POUs/Safety/Components/Euchner_MGB2/Structure/MSM/ST_Euchner_MSM_HW_IN.TcDUT
TYPE ST_Euchner_MSM_HW_IN :
STRUCT
	///Hardware In
	nByte0: USINT;
END_STRUCT
END_TYPE

// ---- POUs/Safety/Components/Euchner_MGB2/Structure/MSM/ST_Euchner_MSM_HW_OUT.TcDUT
TYPE ST_Euchner_MSM_HW_OUT :
STRUCT
	///Hardware Out
	nByte0: USINT;
END_STRUCT
END_TYPE

// ---- POUs/Safety/Components/Euchner_MGB2/Structure/MSM/ST_Euchner_MSM_IN.TcDUT
TYPE ST_Euchner_MSM_IN :
STRUCT
	///SM_I_S1 | Nothalt
	bSM_I_S1: BOOL;
	///SM_I_S2 | Taster beleuchtet
	bSM_I_S2: BOOL;
	///SM_I_S3 | Taster beleuchtet
	bSM_I_S3: BOOL;
	///SM_E_S1 | Fehler Sx
	bSM_E_S1: BOOL;
END_STRUCT
END_TYPE

// ---- POUs/Safety/Components/Euchner_MGB2/Structure/MSM/ST_Euchner_MSM_OUT.TcDUT
TYPE ST_Euchner_MSM_OUT :
STRUCT
	///SM_O_H1 | Led Nothalt
	bSM_O_H1: BOOL;
	///SM_O_H2 | Led Taster S2
	bSM_O_H2: BOOL;
	///SM_O_H3 | Led Taster S3
	bSM_O_H3: BOOL;
	///SM_O_H1 | Led Nothalt blink
	bSM_O_H1_B: BOOL;
	///SM_O_H2 | Led Taster S2 blink
	bSM_O_H2_B: BOOL;
	///SM_O_H3 | Led Taster S3 blink
	bSM_O_H3_B: BOOL;
END_STRUCT
END_TYPE

// ---- POUs/Safety/Components/Euchner_MGB2/Structure/ST_MGB2_IO.TcDUT
TYPE ST_MGB2_IO :
STRUCT
	stHwInMgb				AT%I*	: ST_Euchner_MGB2_HW_IN;
	stHwInMsm				AT%I*	: ST_Euchner_MSM_HW_IN;
	stHwInMsmConfirm		AT%I*	: ST_Euchner_MSM_HW_IN;

	stHwOutMgb				AT%Q*	: ST_Euchner_MGB2_HW_OUT;
	stHwOutMsm				AT%Q*	: ST_Euchner_MSM_HW_OUT;
	stHwOutMsmConfirm		AT%Q*	: ST_Euchner_MSM_HW_OUT;

	/// Door safety ok from Safety plc
	bSAFE_DoorSafetyOk		AT%I*	: BOOL;	
	
	bSAFE_UnlockDoor		AT%Q*	: BOOL;		
END_STRUCT
END_TYPE

// ---- POUs/Safety/Components/SafetyDoor/Structure/ST_SafetyDoor_IN.TcDUT
TYPE ST_SafetyDoor_IN :
STRUCT
	bStartButton : BOOL;
	bRequestButton : BOOL;
	bLockButton : BOOL;
	bLocked : BOOL;
	tsSafe : BOOL;
	tsOpen : BOOL;
	tsSegment_Open : BOOL;
END_STRUCT
END_TYPE

// ---- POUs/Safety/Components/SafetyDoor/Structure/ST_SafetyDoor_IO.TcDUT
TYPE ST_SafetyDoor_IO :
STRUCT
	stHwIn AT%I* : ST_SafetyDoor_IN;
	stHwOut	AT%Q* : ST_SafetyDoor_OUT;
END_STRUCT
END_TYPE

// ---- POUs/Safety/Components/SafetyDoor/Structure/ST_SafetyDoor_OUT.TcDUT
TYPE ST_SafetyDoor_OUT :
STRUCT
	bStartLight : BOOL;	
	bStopLight : BOOL;	
	bLockLight : BOOL;	
	tsRestart : BOOL;    
	tsLockCmd : BOOL;
	tsLocked : BOOL;
END_STRUCT
END_TYPE

// ---- POUs/Safety/Enumerations/E_EDM_Out.TcDUT
//{attribute 'qualified_only'}
//{attribute 'strict'}
TYPE E_EDM_Out :
(
	eEdmOut_none := 0,										(* Sicherheit | Rückmeldung | Xxx *)
	eEdmOut_Nothalt,

(*Maximum*)
	eEdmOut_nMaxIdx
);
END_TYPE

// ---- POUs/Safety/Enumerations/E_Safety_Actor.TcDUT
//{attribute 'qualified_only'}
//{attribute 'strict'}
TYPE E_Safety_Actor :
(
	eSafety_Actor_none := 0,										(* Sicherheit | Rückmeldung | Xxx *)
	eSafety_Actor_NotHalt,
	eSafety_Actor_Freigabeventil_Area1,
	eSafety_Actor_NotHalt_Extern,

(*Maximum*)
	eSafety_Actor_nMaxIdx
);
END_TYPE

// ---- POUs/Safety/Enumerations/E_EmergencyStop.TcDUT
//{attribute 'qualified_only'}
//{attribute 'strict'}
TYPE E_EmergencyStop :
(
	eEmergencyStop_none := 0,
	eEmergencyStop_1 := 1,		// ES1
	eEmergencyStop_2 := 2,		// ES2

	eEmergencyStop_nMaxIdx	
);
END_TYPE

// ---- POUs/Safety/Enumerations/E_Door.TcDUT
//{attribute 'qualified_only'}
//{attribute 'strict'}
TYPE E_Door :
(
	eDoor_none := 0,
	
	eDoor_nMaxIdx	
);
END_TYPE

// ---- POUs/Safety/Structures/Diag/E_HistoryDiagDevices.TcDUT
{attribute 'qualified_only'}
{attribute 'strict'}
TYPE E_HistoryDiagDevices :
(
	EL19xx		:= 0,
	EL29xx 		:= 1
);
END_TYPE

// ---- POUs/Safety/Structures/Diag/ST_DiagHistory.TcDUT
TYPE ST_DiagHistory :
STRUCT
	nMaximum_Messages: BYTE;
	nNewest_Message: BYTE;
	nNewest_Acknowledged_Message: BYTE;
	bNewMessagesAvailable: BOOL;
	nFlags: UINT;
	DiagMessages: ARRAY[1..64] OF ST_DiagMessage;
END_STRUCT
END_TYPE

// ---- POUs/Safety/Structures/Diag/ST_DiagMessage.TcDUT
TYPE ST_DiagMessage :
STRUCT
	nDiagCode: UDINT;
	nFlags: ST_DiagMessageFlags;
	/// The text defined in the ESI file (//DiagMessages)
	nTextID: UINT;
	nTimeStamp: ULINT;
	aParameter: ARRAY[1..16] OF BYTE;
END_STRUCT
END_TYPE

// ---- POUs/Safety/Structures/Diag/ST_DiagMessageFlags.TcDUT
TYPE ST_DiagMessageFlags :
STRUCT
	bInfo: BIT;
	bWarning: BIT;
	bError: BIT;
	bReserved1: BIT;
	bIsLocalTimeStampOfSlave: BIT;
	bReserved2: BIT;
	bReserved3: BIT;
	bReserved4: BIT;
	NumOfParamsInDiagMessage: BYTE;
END_STRUCT
END_TYPE

// ---- POUs/Safety/Structures/Diag/ST_ELM3xxxPAIInfoData.TcDUT
TYPE ST_ELM3xxxPAIInfoData :
STRUCT
	nCPU_Usage: UINT;
	nDeviceState: UINT;
	nOperating_Time: UDINT;
	nOverTemperature_Time: UDINT;
	fDeviceTemperature: REAL;
	fDeviceTemperatureMin: REAL;
	fDeviceTemperatureMax: REAL;
END_STRUCT
END_TYPE

// ---- POUs/Safety/Structures/Diag/ST_MessageItem.TcDUT
TYPE ST_MessageItem :
STRUCT
	/// time stamp
	dtTimeStamp: DT;
	/// priority info, warning, error
	nPriority: BYTE;
	/// message string
	sMessage: T_MaxString;
END_STRUCT
END_TYPE

// ---- POUs/Safety/Structures/Diag/ST_SafetyDiagInfo.TcDUT
TYPE ST_SafetyDiagInfo :
STRUCT
	usintState			:USINT;
	usintDummy			:USINT;
	uintDiag			:UINT;
	usintDiag			:USINT;
END_STRUCT
END_TYPE

// ---- POUs/Safety/Structures/ST_SafetyIn.TcDUT
TYPE ST_SafetyIn :
STRUCT
	/// general safety info
	nProjectCrc				: WORD;
	nSerialNumber			: UDINT;
	
	/// EmergencyStop/Not-Halt von Safety
	bSAFE_ES_Ok				: BOOL;
	
	/// Safe areas sum from safety
	bSAFE_Areas_Ok			: BOOL;
	
	bSAFE_Area_Ok_ST10,
	bSAFE_Area_Ok_ST20,
	
	bSAFE_ConfirmTimeout	: BOOL;
	
	bSAFE_EStop_State		: ARRAY[0..E_EmergencyStop.eEmergencyStop_nMaxIdx] OF BOOL;	(*	state of every emergency stop button	*)
	
	/// safety area OK from safety
	bSAFE_AREA_Ok			: ARRAY[0..iSafety_Anzahl_Schutzbereiche] OF BOOL;
	/// feeedback safety are switched off from safety
	bSafetyAreaSwitchedOff	: ARRAY[0..iSafety_Anzahl_Schutzbereiche] OF BOOL;
	
	/// GATE OK von Safety
	bSAFE_GATE_Ok			: ARRAY[0..E_Door.eDoor_nMaxIdx] OF BOOL;
			
	/// Zustimmeinrichtung von Safety
	bCompressedAirOk		: BOOL;
	
	bSAFE_DRIVES_STO,
	bSAFE_DRIVE_A_STO,
	bSAFE_DRIVE_B_STO,
	bSAFE_DRIVES_HG_STO		: BOOL;
	
	//------------------------------------------------------------------------------------------------------------
	//user definged variables
	
	bSafe_OpMode_Off,
	bSafe_OpMode_Manual,
	bSafe_OpMode_Ruest,
	bSafe_OpMode_Auto				: BOOL;
	
	bSafe_EL6900_WcState				: ARRAY[0..iSafety_Anzahl_EL69xx] OF BOOL; 	(* 	Eingang FB TwinSAFE WcState	*)
	bSafe_FbError_Master				: ARRAY[0..iSafety_Anzahl_TwinSafeGruppen] OF BOOL; 	(* 	Eingang FB TwinSAFE Error -> Safety Master Klemme	*)
	bSafe_ComError_Master				: ARRAY[0..iSafety_Anzahl_TwinSafeGruppen] OF BOOL; 	(* 	Eingang Com TwinSAFE Error -> Safety Master Klemme	*)
	bSafe_OutError_Master				: ARRAY[0..iSafety_Anzahl_TwinSafeGruppen] OF BOOL; 	(* 	Eingang Out TwinSAFE Error -> Safety Master Klemme	*)
	bSafe_OtherError_Master				: ARRAY[0..iSafety_Anzahl_TwinSafeGruppen] OF BOOL; 	(* 	Eingang OtherError TwinSAFE Error -> Safety Master Klemme	*)
                                                                                
	bSafe_AX5805_Error					: ARRAY[0..E_Axis.eAxis_MaxAxis] OF BOOL;	(*	AX5805 Status	*)	
	bSafety_Aktor						: ARRAY[0..100] OF BOOL;		(*	From Safety Logic Aktor	*)
		
END_STRUCT
END_TYPE

// ---- POUs/Safety/Structures/ST_SafetyIO.TcDUT
TYPE ST_SafetyIO :
STRUCT
	stIn	AT%I* : ST_SafetyIn;
	stOut	AT%Q* : ST_SafetyOut;
END_STRUCT
END_TYPE

// ---- POUs/Safety/Structures/ST_SafetyOut.TcDUT
TYPE ST_SafetyOut :
STRUCT
	/// Restart from PLC
	bRestartPLC		: BOOL;		// Fuer Safety-FBs und AX5805
	
	//------------------------------------------------------------------------------------------------------------
	//user definged variables
	bSafetyErrAck			: ARRAY[0..iSafety_Anzahl_EL69xx] OF BOOL ;	(*	Error Ack Sicherheit  *)
	bSafe_Tsg_Run			: ARRAY[0..iSafety_Anzahl_TwinSafeGruppen] OF BOOL; 	(* 	Ausgang Out TwinSAFE Gruppe Run -> Safety Master Klemme	*)
	bSafety_EDM_OUT			: ARRAY[0..100] OF BOOL;		(* 1 = ES	To Safety Logic EDM	*)
	
	bSAFE_LockCmdA,
	bSAFE_LockCmdB			: BOOL;
END_STRUCT
END_TYPE

// ---- POUs/Plant/ST010_OvenA/_Enumerations/E_St010_Settings.TcDUT
//{attribute 'qualified_only'}
//{attribute 'strict'}
{attribute 'to_string'}
{attribute 'to_wstring'}
TYPE E_St010_Settings :
(
	//eSt010_Settings_none := 0,
	
	eSt010_Settings_Station_Deaktiv,	// Station deaktivieren
	eSt010_Settings_Autohome,			// automatic home with start button
	
	eSt010_Settings_HomeSpeed,			// Homing-Geschwindigkeit [mm/s]
	eSt010_Settings_JogSpeed,			// Tippgeschwindigkeit [mm/s]
	eSt010_Settings_WorkSpeed,			// Automatik-Geschwindigkeit [mm/s]
	eSt010_Settings_JogSpeedCh,			// Tippgeschwindigkeit CH-Achsen [mm/s]
	eSt010_Settings_WorkSpeedCh,		// Automatik-Geschwindigkeit CH-Achsen [mm/s]

	eSt010_Settings_AxisRefPos,			// Referenzposition Achse [mm]
	eSt010_Settings_PosHome,			// Homeposition [mm]
	eSt010_Settings_PosWork,			// Mitnehmerposition unteres Segment [mm]
	
	eSt010_Settings_PosHomeCh,			// Homeposition CH-Achsen [mm]
	eSt010_Settings_PosWorkCh,			// Arbeitsposition CH-Achsen [mm]
	
	eSt010_Settings_OvenFixPartHeight,	// Festteilhöhe [mm]
	eSt010_Settings_OvenSegmentHeight,	// Festteilhöhe [mm] //366
	
	eSt010_Settings_OvenMiddlePointX,	// Mittelpunnkt in X-Richtung [mm]
	eSt010_Settings_OvenOffsetY,		// Y-Offset Ofen [mm]
	eSt010_Settings_OvenPickUpDepthZ,	// Teach-Position, Storage 2 Z [mm]
	
	eSt010_Settings_XPosRp1,			// Teach-Position, Ofen A, RP 1 X [mm]
	eSt010_Settings_YPosRp1,			// Teach-Position, Ofen A, RP 1 Y [mm]
	eSt010_Settings_ZPosRp1,			// Teach-Position, Ofen A, RP 1 Z [mm]
	                                                            
	eSt010_Settings_XPosRp2,			// Teach-Position, Ofen A, RP 2 X [mm]
	eSt010_Settings_YPosRp2,			// Teach-Position, Ofen A, RP 2 Y [mm]
	eSt010_Settings_ZPosRp2,			// Teach-Position, Ofen A, RP 2 Z [mm]
	
	/// has to be set to last index for array bounds!
	eSt010_Settings_nMaxIdx
);
END_TYPE

// ---- POUs/Plant/ST010_OvenA/_Structures/ST_St010_HMI_OUT.TcDUT
TYPE ST_St010_HMI_OUT :
STRUCT
	//Trolley	: ST_Trolley;
END_STRUCT
END_TYPE

// ---- POUs/Plant/ST010_OvenA/_Structures/ST_St010_IO_IN.TcDUT
TYPE ST_St010_IO_IN :
STRUCT	
	// inputs
	bRefpos	: BOOL;	// Sensor | Oven | Referenzposition | BMK: =P260+xyz- | Terminal: .: | Tc3Hmi
	
END_STRUCT
END_TYPE

// ---- POUs/Plant/ST010_OvenA/_Structures/ST_St010_IO.TcDUT
TYPE ST_St010_IO :
STRUCT
	stIn 	AT%I* : ST_St010_IO_IN;
	stOut 	AT%Q* : ST_St010_IO_OUT;
	
	stHeatingPlateIO : ST_FurnaceIO;
END_STRUCT
END_TYPE

// ---- POUs/Plant/ST010_OvenA/_Structures/ST_St010_IO_OUT.TcDUT
TYPE ST_St010_IO_OUT :
STRUCT
	bOvenFan :BOOL;
END_STRUCT
END_TYPE

// ---- POUs/Plant/_Structures/ST_MODULE_STATIONS_INFO.TcDUT
// info struct for module stations
TYPE ST_MODULE_STATIONS_INFO :
STRUCT
	bStation_All_Auto 			: BOOL;
	bStation_Any_Manual 		: BOOL;
	bStation_Any_Step 			: BOOL;
	bStation_Any_Error 			: BOOL;	
	bStation_Any_Warning 		: BOOL;	
	bStation_Any_Info 			: BOOL;	
	
	bStation_All_Started 		: BOOL;
	bStation_All_Stopped		: BOOL;
	bStation_All_InHome 		: BOOL;
	bStation_Any_Homing 		: BOOL;
END_STRUCT
END_TYPE

// ---- POUs/Plant/_Structures/ST_MODULES_INFO.TcDUT
// info struct for all modules
TYPE ST_MODULES_INFO EXTENDS ST_MODULE_STATIONS_INFO :
STRUCT
	astModuleStationsInfo	: ARRAY[0..E_Module.eModule_nMaxIdx] OF ST_MODULE_STATIONS_INFO;
END_STRUCT
END_TYPE

// ---- POUs/System/Supervision/Enumerations/Alarmsystem/E_AlarmPriority.TcDUT
{attribute 'qualified_only'}
{attribute 'strict'}
{attribute 'to_string'}
TYPE E_AlarmPriority :
(
	Undefined 	:= 0,
	Info 		:= 1,
	Warning 	:= 2,
	Error 		:= 3
);
END_TYPE

// ---- POUs/System/Supervision/Enumerations/Alarmsystem/E_AlarmState.TcDUT
{attribute 'qualified_only'}
{attribute 'strict'}
{attribute 'to_string'}
/// Enum for the Alarm states
TYPE E_AlarmState :
( 
	/// Undefined, not init state
	Undefined 	:= 0,
	/// Alarm is inactive
	Inactive 	:= 1,
	/// Alarm is active (raised)
	Active 		:= 2,
	/// Alarm is ack
	Ack 		:= 3	
);
END_TYPE

// ---- POUs/System/Supervision/Enumerations/Alarmsystem/E_EventReaction.TcDUT
{attribute 'qualified_only'}
{attribute 'strict'}
{attribute 'to_string'}
TYPE E_EventReaction :
(
	Undefined 			:= 0,
	NoReaction 			:= 1,
	CycleStop			:= 11,
	Stop 				:= 21,
	Init				:= 31
);
END_TYPE

// ---- POUs/System/Supervision/Enumerations/E_EtherCatBox.TcDUT
/// enumeration of all possible EC Boxes
TYPE E_EtherCatBox :
(
	eEtherCatBox_ControlCabinet := 0,
	eEtherCatBox_Oven_A := 1,
	eEtherCatBox_Oven_B := 2,
	eEtherCatBox_Storage := 3,
	
	eEtherCatBox_nMaxIdx
);
END_TYPE

// ---- POUs/System/Supervision/EtherCAT/Enumerations/E_EcDeviceState.TcDUT
/// Enumeration of possible EtherCAT states.
TYPE E_EcDeviceState :
(
	/// no error
	eEtherCATState_NoError := 0,
	/// Link error
	eEtherCATState_LinkError := 16#1,
	/// I/O locked after link error (I/O reset required)
	eEtherCATState_IoLockedAfterLinkErr := 16#2,
	/// Link error (redundancy adapter)
	eEtherCATState_LinkErrRedAdapter := 16#4,
	/// Missing one frame (redundancy mode)
	eEtherCATState_MissingFrame := 16#8,
	/// Out of send resources (I/O reset required)
	eEtherCATState_OutOfSendResources := 16#10,
	/// Watchdog triggered
	eEtherCATState_WatchdogTriggered := 16#20,
	/// Ethernet driver (miniport) not found
	eEtherCATState_EthernetDrvNotFound := 16#40,
	/// I/O reset active
	eEtherCATState_IO_resetActive := 16#80,
	/// At least one device in 'INIT' state
	eEtherCATState_AtLeastOneDeviceInit := 16#100,
	///  At least one device in 'PRE-OP' state
	eEtherCATState_AtLeastOneDevicePreOp := 16#200,
	/// At least one device in 'SAFE-OP' state
	eEtherCATState_AtLeastOneDeviceSafeOp := 16#400,
	/// At least one device indicates an error state
	eEtherCATState_AtLeastOneDeviceError := 16#800,
	/// DC not in sync
	eEtherCATState_DC_notInSync := 16#1000
);
END_TYPE

// ---- POUs/System/Supervision/Structures/ST_EcMaster_In.TcDUT
TYPE ST_EcMaster_In :
STRUCT
	/// AmsNetId of EtherCAT device
	stAmsAdr 						:ST_AmsAddr;
	/// DeviceId of EtherCAT device
	nDevId							:UINT;
	/// Device state of EtherCAT device
	nDeviceState					:UINT;
END_STRUCT
END_TYPE

// ---- POUs/System/Supervision/Structures/ST_GridObject_Register.TcDUT
TYPE ST_GridObject_Register :
STRUCT
	sGroup				:STRING;
	dtZeitStempel		:STRING;
	fFuelldruck			:REAL;
	fFuellzeit			:REAL;
	fGasTemperatur		:REAL;	
	fLaenge_Mit_Kappe	:REAL;
	fLaenge_Ohne_Kappe	:REAL;
	fMasse_Differenz	:REAL;
	fMasse_Leer			:REAL;	
	fMasse_Voll			:REAL;
	ePartState			:STRING;	
END_STRUCT
END_TYPE

// ---- POUs/System/Supervision/Structures/ST_SystemVars.TcDUT
TYPE ST_SystemVars :
STRUCT
	/// global program cycle counter
	nStepCounter				:UDINT;
	
	/// path of the actual method
	wsActualMethod				:WSTRING(255);
	
	/// current system time
	dtNow						:DT;
	stNow						:TIMESTRUCT;
	
	/// current system time in string format	
	sTimeString					:STRING;
	
	/// PLC system informations
	stPlcSystemInfo				:ST_PlcSystemInfo;
	
	/// default pulse struct
	stPulse						:ST_DefaultPulse;
		
	/// Default epsilon (e.g.: positioning window)
	fEpsilon					:LREAL := 1E-5;
	/// Empty string value
	sEmpty						:STRING(1);

END_STRUCT
END_TYPE

// ---- POUs/System/Utilities/Counter/E_Counter.TcDUT
//{attribute 'qualified_only'}
//{attribute 'strict'}
TYPE E_Counter :
(
	eCounter_General,	//Allgemein
	//eCounter_Maintenance,	//Wartung
	eCounter_Shift,		//Schicht Zaheler
	//eCounter_Order,		//Auftrag Zaheler	
	//eCounter_St001,		//Station 001
	//eCounter_St002,		//Station 002
	//eCounter_St003,		//Station 003
	//eCounter_St004,		//Station 004
	//eCounter_St005,		//Station 005
	//eCounter_St006,		//Station 006
	//eCounter_St007,		//Station 007
	//eCounter_St008,		//Station 008
	//eCounter_St009,		//Station 009
	//eCounter_St010,		//Station 010
	//eCounter_St011,		//Station 011
	//eCounter_St012,		//Station 012
	//eCounter_St013,		//Station 013
	//eCounter_St014,		//Station 014
	//eCounter_St015,		//Station 015
	//eCounter_St016,		//Station 016
	//eCounter_St017,		//Station 017
	//eCounter_St018,		//Station 018
	//eCounter_St100,		//Station 100
	
	eCounter_Max
);
END_TYPE

// ---- POUs/System/Utilities/Counter/E_CounterMode.TcDUT
{attribute 'qualified_only'}
{attribute 'strict'}
TYPE E_CounterMode :
(
	eCounterMode_none := 0,
	eCounterMode_Ok_Up,
	eCounterMode_Ok_Down,
	eCounterMode_Nok_Up,
	eCounterMode_Nok_Down,	
	eCounterMode_Ok_Clear,
	eCounterMode_Nok_Clear,
	eCounterMode_SerialError_Clear,
	eCounterMode_All_Clear	
);
END_TYPE

// ---- POUs/System/Utilities/Counter/ST_Counter_Item.TcDUT
TYPE ST_Counter_Item :
STRUCT
	stIndex						: ST_Text;
	stGroup						: ST_Text;
	stName						: ST_Text;
	nValueOk					: DINT;	
	nValueNok					: DINT;
	nValueTotal					: DINT;
	nValueSerialError			: DINT;
	nValueOkLevel1				: DINT;
	eReactionOkLevel1			: E_CounterReaction;
	nValueOkLevel2				: DINT;
	eReactionOkLevel2			: E_CounterReaction;
	nValueNokLevel1				: DINT;
	eReactionNokLevel1			: E_CounterReaction;
	nValueNokLevel2				: DINT;
	eReactionNokLevel2			: E_CounterReaction;
	nValueTotalLevel1			: DINT;
	eReactionTotalLevel1		: E_CounterReaction;
	nValueTotalLevel2			: DINT;
	eReactionTotalLevel2		: E_CounterReaction;	
	eUserLevel					: E_User_Level;
	eDataType					: E_DataType;
                                  
	eCurrentReactionOkLevel1	: E_CounterReaction;
	eCurrentReactionOkLevel2	: E_CounterReaction;
	eCurrentReactionNokLevel1	: E_CounterReaction;	
	eCurrentReactionNokLevel2	: E_CounterReaction;
	eCurrentReactionTotalLevel1	: E_CounterReaction;
	eCurrentReactionTotalLevel2	: E_CounterReaction;	
	                              
	eCurrentCounterState		: E_CounterReaction;	
END_STRUCT
END_TYPE

// ---- POUs/System/Utilities/CSV/Structures/ST_FillOrder.TcDUT
TYPE ST_FillOrder :
STRUCT
	bActive		: BOOL;
	//dtTimeStamp	: DT;
	//eLevel		: E_LogLevel;
	//sSource		: STRING(31);
	//sMessage 	: T_MaxString;
END_STRUCT
END_TYPE

// ---- POUs/System/Utilities/Var2File/Structures/ST_Var2File_Com.TcDUT
/// Communication structure to the Var2File application 
TYPE ST_Var2File_Com :
STRUCT
	// FROM Application
	
	/// Application is running (application set to 1000 every 1 sec) 
	nAppRunning				: UDINT;
	
	/// Application work progress
	nAppProgress			: UDINT;

	/// Applications error code
	nAppErrorCode			: UDINT;
	
	/// App-Job ist finished
	bAppJobFinished			: BOOL;
	
	/// App-Job canceled by user
	bAppJobCanceled			: BOOL;
	
	
	// TO Application
	/// request job cancel
	bJobCancelRequest		: BOOL;
END_STRUCT
END_TYPE

// ---- POUs/System/Utilities/Var2File/Structures/ST_Var2File_Config.TcDUT
TYPE ST_Var2File_Config :
STRUCT
	/// Path to Var2File exe
	sAppExeFilePath		: STRING(255) := '/usr/local/var2file/';
	
	/// Var2File exe name
	sAppExeFileName		: STRING(25) := 'Var2File.Core.App.dll';
	
	/// Filterset number for all variables
	nFilterSetIDAllVars		: INT := 2;
	
	/// Default path for Var2File data 
	sDefaultFileFolderPath	: STRING(255) := '/usr/local/var2file/data';
	
	/// NetId
	sAmsNetId				: STRING := '';
END_STRUCT
END_TYPE

// ---- GVLs/CONST.TcGVL
/// Global constants
//{attribute 'qualified_only'}
VAR_GLOBAL CONSTANT
	sVersion				: STRING := 'Version 0.1';

	/// debug logging source const
	sSource					: STRING(10) := 'Machine';
	
	/// zero based max indexes
	iMaxIdxEcMaster			: INT := 0;		// max index of EtherCAT master
	
	iMaxIdxUnitTest			: INT := 1;		// max index of unit test
	iMaxIdxSystemInfo		: INT := 30;	// max index of system info
	iMaxIdxRecipe			: INT := 50;	// max index of recipe
	
	iMaxIdxLocalSetting		: INT := 100;	// max index of plant-, module- or station-setting
	iMaxIdxLocalStepChain	: INT := 1;		// max index of plant-, module- or station-step chain
	iMaxIdxLocalButton		: INT := 20;	// max index of plant-, module- or station-button (HMI)
	iMaxIdxObject			: INT := 20;	// max index of plant-, module- or station-object
	iMaxIdxMonitoring		: INT := 50;	// max index of plant-, module-, station- or object monitoring
	iMaxIdxCounter			: INT := 1;		// max index of counter (0 = total, 1 = day, 2..n = station)
	
	iMaxIdxAlam				: INT := 100;	// max index of alarm item
	iMaxIdxNoti				: INT := 150;	// max index of notification item
	iMaxIdxNotiArchiv		: INT := 300;	// max index of notification archiv item
	
	iMaxIdxLayout			: INT := 3;		// max index of possible layouts
	
	iMaxIdxPalletWorkpieceX	: INT := 6;		// max index of pallet-workpiece X
	iMaxIdxPalletWorkpieceY	: INT := 8;		// max index of pallet-workpiece Y
	
	iMaxIdxTrolleyPalletX	: INT := 1;		// max index of trolley-pallet X
	iMaxIdxTrolleyPalletY	: INT := 19;	// max index of trolley-pallet Y
	
	iMaxIdxStoragePallet	: INT := 1;		// max index of storage-pallet
	
	// global text list
	stTextListGlobal		: ST_Text_List_Global;
	
	wsEmpty					: WSTRING := "";
	stEmptyText				: ST_Text := (nNameId := 0, wsNameId := "", wsName := "");
	stEmptyDataItem			: ST_Data_Item;
	
	chAxisPosTol 			: LREAL := 3;
	lreal_max 				: LREAL := 1.797E308;  // LREAL max
	
	bEnSafetyOpMode			: BOOL := FALSE;
	sDirSeparator			: STRING(1) := '/'; // for TcBsd: /, for Windown: '\'
END_VAR

(*	Safety Konstanten	*)
VAR_GLOBAL CONSTANT
	{attribute 'const_non_replaced'}
	stLibVersion_PLC 						: ST_LibVersion := (iMajor := 1, iMinor := 0, iBuild := 0, iRevision := 0, nFlags := 0, sVersion := '1.0');
	
	iSafety_Anzahl_EL69xx					: INT := 1;	(*	Anzahl an TwinSAFE Logikklemmen im System	*)
	iSafety_Anzahl_TwinSafeGruppen			: INT := 1;	(*	Anzahl an Gruppen in einer TwinSAFE Logikklemmen	*)
	iSafety_Anzahl_Schutzbereiche			: INT := 2;	(*	Anzahl an Schutzbereiche (Einlauf, Bearbeitung, Auslauf, ...)	*)

	(*	Diagnose	*)
	iSafetyDiag_Anzahl_FbEmergencyStop		: INT := 20;	(*	Anzahl an NotHalt Bausteindiagnosen	*)
	iSafetyDiag_Anzahl_FbMachineMonitoring	: INT := 20;	(*	Anzahl an Maschine Monitoring Bausteindiagnosen	*)
	iSafetyDiag_Anzahl_FbTwoHand			: INT := 50;	(*	Anzahl an 2Hand Bausteindiagnosen	*)
	iSafetyDiag_Anzahl_FbEDM				: INT := 10;	(*	Anzahl an 2Hand Bausteindiagnosen	*)
END_VAR

// ---- GVLs/GVL.TcGVL
/// Project specific global var's
//{attribute 'qualified_only'}
VAR_GLOBAL
	// ToDo: comissioning
	iIBN : INT := 1;
	bTest : BOOL;
END_VAR

// ---- GVLs/HMI.TcGVL
/// HMI var's
//{attribute 'qualified_only'}
VAR_GLOBAL
	
	// current user level
	eUserLevel				: E_User_Level;

	/// HMI IOs
	stHmi					: ST_HMI;				// PLC internal HMI usage (HMI summary)
	stHmiInOut				: ST_HMI_InOut;			// direct HMI IN OUT access
	
	stHmiHw					: HMI_PROVIDER_HW_IO;	// HW Pult IOs
	stHmiTc3				: ST_Hmi_Tc3; 			// TC3 HMI interface
	
	/// HMI provider
	fbHmiHwProvider			: FB_HMI_PROVIDER_HW;
	fbHmiTc3Provider		: FB_HMI_Provider_TC3;
END_VAR

VAR_GLOBAL PERSISTENT
	// actual language
	eLanguage			: E_Language := E_Language.DE;
	
	// counter	            
	stCounter			: ARRAY[0..CONST.iMaxIdxCounter] OF ST_Counter_Item;
	stOverallCounter	: ST_Counter;
	stShiftCounter		: ST_Counter;
END_VAR

// ---- GVLs/IO.TcGVL
/// Machine IO structures 
{attribute 'qualified_only'}
VAR_GLOBAL
	
	/// Safety IO'S
	stSafetyIO			: ST_SafetyIO;
	
	/// control cabinet IOs
	stControlCabinetIO	: ST_ControlCabinetIO;
	
	// module
	stM001_Module_IO	: ST_M001_IO;

	// stations
	{attribute 'contextName' := 'PlcTask'}
	st010_OvenA_IO		: ST_St010_IO;
	{attribute 'contextName' := 'PlcTask'}
	st020_OvenB_IO		: ST_St020_IO;
	{attribute 'contextName' := 'PlcTaskFast'}
	st030_Handling_IO	: ST_St030_IO;
	{attribute 'contextName' := 'PlcTask'}
	st040_Storage_IO	: ST_St040_IO;
	{attribute 'contextName' := 'PlcTask'}
	st050_Mould_IO		: ST_St050_IO;

	
END_VAR

// ---- GVLs/NcIO.TcGVL
{attribute 'qualified_only'}
VAR_GLOBAL
	{attribute 'contextName' := 'PlcTask'}
//	{attribute 'TcNcAxis' := 'AxisTest'}
//	stAxisTest					: AXIS_REF;
//	{attribute 'contextName' := 'PlcTask'}
//	stAxisTestIO				: ST_AxisIO;

//  virtual master	
	stAxis_VirtualMaster		: AXIS_REF;
	stAxis_VirtualMaster_IO		: ST_AxisIO;

//  ST010 OvenA	
	stAxis_ST010_OvenA			: AXIS_REF;
	stAxis_ST010_OvenA_IO		: ST_AxisIO;
	
	stAxis_ST010_OvenACh1		: AXIS_REF;
	stAxis_ST010_OvenACh1_IO	: ST_AxisIO;
	
	stAxis_ST010_OvenACh2		: AXIS_REF;
	stAxis_ST010_OvenACh2_IO	: ST_AxisIO;
	
//  ST020 OvenB
	stAxis_ST020_OvenB			: AXIS_REF;
	stAxis_ST020_OvenB_IO		: ST_AxisIO;
	
	stAxis_ST020_OvenBCh1		: AXIS_REF;
	stAxis_ST020_OvenBCh1_IO	: ST_AxisIO;
	
	stAxis_ST020_OvenBCh2		: AXIS_REF;
	stAxis_ST020_OvenBCh2_IO	: ST_AxisIO;
	
//  ST030 Handling
	stAxis_ST030_AxisX			: AXIS_REF;
	stAxis_ST030_AxisX_IO		: ST_AxisIO;
	
	stAxis_ST030_AxisY			: AXIS_REF;
	stAxis_ST030_AxisY_IO		: ST_AxisIO;
	
	stAxis_ST030_AxisZ			: AXIS_REF;
	stAxis_ST030_AxisZ_IO		: ST_AxisIO;
	
//  ST040 Storage
	stAxis_ST040_Axis1			: AXIS_REF;
	stAxis_ST040_Axis1_IO		: ST_AxisIO;
	
	stAxis_ST040_Axis2			: AXIS_REF;
	stAxis_ST040_Axis2_IO		: ST_AxisIO;
	

	stAxisDummy					: AXIS_REF;
END_VAR

// ---- GVLs/Safety.TcGVL
//{attribute 'qualified_only'}
VAR_GLOBAL

(*	Diagnose Safety PLC		*)
	Iarr_SafetyDiag_NotHalt					AT %I*	:ARRAY[0..iSafetyDiag_Anzahl_FbEmergencyStop] OF ST_SafetyDiagInfo;	(*	Safety Diagnose Info für Not-Halt Baustein		*)
	fbDiag_NotHalt									:ARRAY[0..iSafetyDiag_Anzahl_FbEmergencyStop] OF FB_TwinSAFEDiag_EmergencyStop;
	Iarr_SafetyDiag_MachineMonitoring		AT %I*	:ARRAY[0..iSafetyDiag_Anzahl_FbMachineMonitoring] OF ST_SafetyDiagInfo;	(*	Safety Diagnose Info für Schutztüren Baustein		*)
	fbDiag_MachineMonitoring						:ARRAY[0..iSafetyDiag_Anzahl_FbMachineMonitoring] OF FB_TwinSAFEDiag_MachineMonitoring;
	Iarr_SafetyDiag_TwoHand					AT %I*	:ARRAY[0..iSafetyDiag_Anzahl_FbTwoHand] OF ST_SafetyDiagInfo;	(*	Safety Diagnose Info für 2Hand Baustein		*)
	fbDiag_TwoHand									:ARRAY[0..iSafetyDiag_Anzahl_FbTwoHand] OF FB_TwinSAFEDiag_TwoHand;
	Iarr_SafetyDiag_EDM						AT %I*	:ARRAY[0..iSafetyDiag_Anzahl_FbEDM] OF ST_SafetyDiagInfo;	(*	Safety Diagnose Info für EDM Baustein		*)
	fbDiag_EDM										:ARRAY[0..iSafetyDiag_Anzahl_FbEDM] OF FB_TwinSAFEDiag_EDM;

(*	HW		*)
	fbTwinSAFE_HW_Diag						: ARRAY[1..iSafety_Anzahl_EL69xx] OF FB_TwinSAFE_HW_Diag;
	
	arrSaftyDoors							: ARRAY[0..1] OF ST_SafetyDoor_IO;
END_VAR

// ---- GVLs/Services.TcGVL
//{attribute 'qualified_only'}
VAR_GLOBAL
	b1stShot			: BOOL := TRUE;
	bPlcInitDone,
	bSettingsSaved		: BOOL;
	
	ILog				: I_Logger;
	fbEventHandler		: FB_EventHandler;
	
	fbRecipeManager		: FB_RecipeManager;
	fbVar2File			: FB_Var2File;
	stGlobalModuleInfo	: ST_MODULES_INFO; // global module/staion info
END_VAR
VAR_GLOBAL PERSISTENT
	// current system/machine configuration
	stConfig 			: ST_Configuration;
	
	// settings/recipe            
	stSettings			: ST_Settings;
	
	// PLC app system info
	stPlcAppSystemInfo	: PlcAppSystemInfo;
END_VAR

// ---- GVLs/Plant.TcGVL
//{attribute 'qualified_only'}
VAR_GLOBAL
	// objects (plant-, module- and station objects) 
	stObjects			: ST_Objects;
	
	// modules
	fbModul001			: FB_M001_Module;
	stM001IModule		: ST_M001_Interface;
	
	/// stations
	fbSt010OvenA		: FB_St010_OvenA;
	stSt010IOvenA		: ST_St010_Interface;
	
	fbSt020OvenB		: FB_St020_OvenB;
	stSt020IOvenB		: ST_St020_Interface;
	
	fbSt030Handling		: FB_St030_Handling;
	stSt030IHandling	: ST_St030_Interface;
	
	fbSt040Storage		: FB_St040_Storage;
	stSt040IStorage		: ST_St040_Interface;
	
	fbSt050Mould		: FB_St050_Mould;
	stSt050IMould		: ST_St050_Interface;
END_VAR

// ---- Background/UnitTest/Interfaces/ITestCase.TcIO
INTERFACE ITestCase

{attribute 'object_name' := 'Reset'}
METHOD Reset
END_METHOD

{attribute 'object_name' := 'Run'}
METHOD Run : E_TestCaseState
END_METHOD

PROPERTY TestResult : E_TestResult
GET
END_GET
END_PROPERTY

PROPERTY TestState : E_TestCaseState
GET
END_GET
END_PROPERTY

END_INTERFACE

// ---- POUs/Components/AxisDriver/Interfaces/ITFMotionComponent.TcIO
INTERFACE ITFMotionComponent EXTENDS ITFComponent

END_INTERFACE

// ---- POUs/Components/_Base/Interfaces/I_ManualUi.TcIO
INTERFACE I_ManualUi

METHOD PUBLIC M_SetStateObject : BOOL
VAR_IN_OUT
	stStateObjectRef : ST_Object_Item;
END_VAR
END_METHOD

PROPERTY Name : ST_Text
GET
END_GET
END_PROPERTY

PROPERTY ObjectIndex : DINT
GET
END_GET
SET
END_SET
END_PROPERTY

END_INTERFACE

// ---- POUs/Components/_Base/Interfaces/ITFComponent.TcIO
INTERFACE ITFComponent EXTENDS __System.IQueryInterface

/// Get's or set's a value indicating whether this component is active or not.
PROPERTY Active : BOOL
GET
END_GET
SET
END_SET
END_PROPERTY

/// Get's value representing the component state.
PROPERTY ClearText : WSTRING(255)
GET
END_GET
END_PROPERTY

PROPERTY ID : INT
GET
END_GET
SET
END_SET
END_PROPERTY

/// Get's value representing the component state.
PROPERTY LastError : T_MaxString
GET
END_GET
END_PROPERTY

PROPERTY Logger : I_Logger
SET
END_SET
END_PROPERTY

PROPERTY Name : ST_Text
GET
END_GET
SET
END_SET
END_PROPERTY

PROPERTY ObjectId : WSTRING
GET
END_GET
END_PROPERTY

PROPERTY Path : String
GET
END_GET
END_PROPERTY

PROPERTY RefsValid : BOOL
GET
END_GET
END_PROPERTY

/// Reset component logic
{attribute 'object_name' := 'Reset'}
METHOD Reset
END_METHOD

/// Run component logic
{attribute 'object_name' := 'Run'}
METHOD Run : E_ComponentState
END_METHOD

/// Get's value representing the component state.
PROPERTY State : E_ComponentState
GET
END_GET
END_PROPERTY

/// Get's value representing the component state.
PROPERTY StateToString : STRING
GET
END_GET
END_PROPERTY

PROPERTY Typ : E_ComponentType
GET
END_GET
END_PROPERTY

END_INTERFACE

// ---- POUs/HMI/Events/Interfaces/I_EventHandler.TcIO
INTERFACE I_EventHandler

METHOD PUBLIC ArgAddDint : I_EventHandler
VAR_INPUT
	value : DINT;
END_VAR
END_METHOD

METHOD PUBLIC ArgAddEventRef : I_EventHandler
VAR_INPUT
	value : TcEventEntry;
END_VAR
END_METHOD

METHOD PUBLIC ArgAddLreal : I_EventHandler
VAR_INPUT
	value : LREAL;
END_VAR
END_METHOD

METHOD PUBLIC ArgAddString : I_EventHandler
VAR_IN_OUT CONSTANT
	value : STRING;
END_VAR
END_METHOD

METHOD PUBLIC ArgAddWString : I_EventHandler
VAR_IN_OUT CONSTANT
	value : WSTRING;
END_VAR
END_METHOD

METHOD PUBLIC ArgClear : I_EventHandler
END_METHOD

METHOD PUBLIC ArgSbAppend : I_EventHandler
VAR_IN_OUT CONSTANT
	value : T_MaxString;
END_VAR
END_METHOD

METHOD PUBLIC ArgSbAppendAny : I_EventHandler
VAR_INPUT
	value : ANY;
END_VAR
END_METHOD

METHOD PUBLIC ArgSbAppendAnyRaise : HRESULT
VAR_INPUT
	value : ANY;
END_VAR
END_METHOD

METHOD PUBLIC ArgSbAppendRaise : HRESULT
VAR_IN_OUT CONSTANT
	value : T_MaxString;
END_VAR
END_METHOD

METHOD PUBLIC ArgSbAppendS : I_EventHandler
VAR_INPUT
	value : T_MaxString := '';
END_VAR
END_METHOD

METHOD PUBLIC ArgSbAppendSet : I_EventHandler
VAR_IN_OUT CONSTANT
	value : T_MaxString;
END_VAR
END_METHOD

METHOD PUBLIC ArgSbAppendWs : I_EventHandler
VAR_IN_OUT CONSTANT
	value : WSTRING;
END_VAR
END_METHOD

METHOD PUBLIC ArgSbAppendWsRaise : HRESULT
VAR_IN_OUT CONSTANT
	value : WSTRING;
END_VAR
END_METHOD

METHOD PUBLIC ArgSbInit : I_EventHandler
VAR_IN_OUT CONSTANT
	value : T_MaxString;
END_VAR
END_METHOD

METHOD PUBLIC ArgSbInitExternal : I_EventHandler
VAR_INPUT
	sb	: I_StringBuilder;
END_VAR
END_METHOD

METHOD PUBLIC ArgSbInitWs : I_EventHandler
VAR_IN_OUT CONSTANT
	value : WSTRING;
END_VAR
END_METHOD

METHOD PUBLIC ArgSetDint : I_EventHandler
VAR_INPUT
	value : DINT;
END_VAR
END_METHOD

METHOD PUBLIC ArgSetEventRef : I_EventHandler
VAR_INPUT
	value : TcEventEntry;
END_VAR
END_METHOD

METHOD PUBLIC ArgSetLreal : I_EventHandler
VAR_INPUT
	value : LREAL;
END_VAR
END_METHOD

METHOD PUBLIC ArgSetSb : I_EventHandler
VAR_INPUT
	sb 		: I_StringBuilder := 0; // optional external string builder, set to 0 to use internal
END_VAR
END_METHOD

METHOD PUBLIC ArgSetSbRaise : HRESULT
VAR_INPUT
	sb	: I_StringBuilder := 0; // optional external string builder, set to 0 to use internal
END_VAR
END_METHOD

METHOD PUBLIC ArgSetString : I_EventHandler
VAR_IN_OUT CONSTANT
	value : STRING;
END_VAR
END_METHOD

METHOD PUBLIC ArgSetWString : I_EventHandler
VAR_IN_OUT CONSTANT
	value : WSTRING;
END_VAR
END_METHOD

METHOD PUBLIC CreateAlarm : I_EventHandler
VAR_INPUT
	stEventEntry      : TcEventEntry;
    bWithConfirmation : BOOL := FALSE;
    ipSourceInfo      : I_TcSourceInfo := NULL;
END_VAR
END_METHOD

PROPERTY ErrorActive : BOOL
GET
END_GET
END_PROPERTY

PROPERTY InfoActive : BOOL
GET
END_GET
END_PROPERTY

METHOD PUBLIC Raise : HRESULT
VAR_INPUT
	nTimeStamp : ULINT := 0;
END_VAR
END_METHOD

METHOD PUBLIC Reset : BOOL
VAR_INPUT
END_VAR
END_METHOD

METHOD PUBLIC Select : I_EventHandler
VAR_INPUT
	stEventEntry : TcEventEntry;
END_VAR
END_METHOD

METHOD PUBLIC Send : BOOL
VAR_INPUT
	stEventEntry      : TcEventEntry;
    ipSourceInfo      : I_TcSourceInfo := NULL;
    nTimeStamp        : ULINT := 0;
    ipArguments       : I_TcArguments := NULL;
END_VAR
END_METHOD

METHOD PUBLIC SendJson : BOOL
VAR_INPUT
	stEventEntry      : TcEventEntry;
    ipSourceInfo      : I_TcSourceInfo := NULL;
    nTimeStamp        : ULINT := 0;
    ipArguments       : I_TcArguments := NULL;
END_VAR
VAR_IN_OUT CONSTANT
    sJsonAttribute    : STRING;
END_VAR
END_METHOD

METHOD PUBLIC SendString : BOOL
VAR_IN_OUT CONSTANT
	msg : STRING;	
END_VAR
END_METHOD

METHOD PUBLIC SendStringJson : BOOL
VAR_IN_OUT CONSTANT
	msg				: STRING;
	sJsonAttribute	: STRING;
END_VAR
END_METHOD

PROPERTY WarningActive : BOOL
GET
END_GET
END_PROPERTY

END_INTERFACE

// ---- POUs/HMI/Provider/_Interfaces/ITF_HMI_PROVIDER.TcIO
INTERFACE ITF_HMI_PROVIDER

PROPERTY ItfHmiIn : REFERENCE TO ST_HMI_IN
GET
END_GET
END_PROPERTY

PROPERTY ItfHmiOut : REFERENCE TO ST_HMI_OUT
GET
END_GET
END_PROPERTY

/// reset
METHOD M_Reset : BOOL
VAR
END_VAR
END_METHOD

METHOD M_Run : BOOL
VAR_INPUT
END_VAR
END_METHOD

PROPERTY Mute : bool
GET
END_GET
END_PROPERTY

PROPERTY Provider : E_HMI_PROVIDER
GET
END_GET
END_PROPERTY

// HMI control request (Bedienhoheit)
//	set ti true, on any control request from the HMI provider (e.g.: watch IN struct)
//	reset will be done by HMI controller, on other provider request  
{attribute 'monitoring' := 'call'}
PROPERTY RequestManualControl : BOOL
GET
END_GET
SET
END_SET
END_PROPERTY

// HMI recipe control request (Bedienhoheit)  
{attribute 'monitoring' := 'call'}
PROPERTY RequestRecipeMgmt : BOOL
GET
END_GET
SET
END_SET
END_PROPERTY

// HMI settings control request (Bedienhoheit)  
{attribute 'monitoring' := 'call'}
PROPERTY RequestSettingMgmt : BOOL
GET
END_GET
SET
END_SET
END_PROPERTY

// HMI user management control request (Bedienhoheit)  
{attribute 'monitoring' := 'call'}
PROPERTY RequestUserMgmt : BOOL
GET
END_GET
SET
END_SET
END_PROPERTY

END_INTERFACE

// ---- POUs/Plant/_Base/Interfaces/IModule.TcIO
INTERFACE IModule EXTENDS ITFComponent

{attribute 'monitoring':='call'}
PROPERTY PUBLIC EmergencyStopOk : BOOL
GET
END_GET
SET
END_SET
END_PROPERTY

METHOD PUBLIC GetStepChainTest : ST_Text
VAR_INPUT
	Index : INT; // step chain index
END_VAR
END_METHOD

PROPERTY InHome : BOOL
GET
END_GET
END_PROPERTY

METHOD Public M_Init : IModule
VAR_INPUT
END_VAR
END_METHOD

METHOD PUBLIC M_InitEvents : IModule
VAR_IN_OUT CONSTANT
	infoEvent,
	warnEvent,
	errorEvent : TcEventEntry;
END_VAR
END_METHOD

METHOD Public M_InitEx : IModule
VAR_INPUT
	ILogger			: I_Logger;
	IEventHandler	: I_EventHandler;
END_VAR
END_METHOD

METHOD PUBLIC M_Run : BOOL
VAR_INPUT
END_VAR
END_METHOD

PROPERTY Module : E_Module
GET
END_GET
SET
END_SET
END_PROPERTY

PROPERTY OpMode : E_OpMode
GET
END_GET
END_PROPERTY

PROPERTY RunCycle : BOOL
GET
END_GET
END_PROPERTY

{attribute 'monitoring':='call'}
PROPERTY PUBLIC SafetyOk : BOOL
GET
END_GET
SET
END_SET
END_PROPERTY

PROPERTY Stopped : BOOL
GET
END_GET
END_PROPERTY

PROPERTY TextAuto : ST_Text
GET
END_GET
END_PROPERTY

PROPERTY TextHome : ST_Text
GET
END_GET
END_PROPERTY

END_INTERFACE

// ---- POUs/Plant/_Base/Interfaces/IStation.TcIO
INTERFACE IStation EXTENDS ITFComponent

PROPERTY PUBLIC Cycles : UDINT
GET
END_GET
SET
END_SET
END_PROPERTY

PROPERTY INTERNAL EmergencyStopOk : BOOL
GET
END_GET
SET
END_SET
END_PROPERTY

PROPERTY INTERNAL Enable : BOOL
GET
END_GET
SET
END_SET
END_PROPERTY

PROPERTY INTERNAL EnableSummary : BOOL
GET
END_GET
END_PROPERTY

METHOD PUBLIC GetStepChainTest : ST_Text
VAR_INPUT
	Index : INT; // step chain index
END_VAR
END_METHOD

{attribute 'monitoring':='call'}
PROPERTY PUBLIC Homing : BOOL
GET
END_GET
END_PROPERTY

PROPERTY InHome : BOOL
GET
END_GET
END_PROPERTY

METHOD PUBLIC InitEvents : IStation
VAR_IN_OUT CONSTANT
	infoEvent,
	warnEvent,
	errorEvent : TcEventEntry;
END_VAR
END_METHOD

METHOD Public M_Init : IStation
VAR_INPUT
END_VAR
END_METHOD

METHOD PUBLIC M_InitEx : IStation
VAR_INPUT
	ILogger			: I_Logger;
	IEventHandler	: I_EventHandler;
END_VAR
END_METHOD

METHOD PUBLIC M_Run : BOOL
VAR_INPUT
END_VAR
END_METHOD

PROPERTY OpMode : E_OpMode
GET
END_GET
END_PROPERTY

PROPERTY Parent : E_Module
GET
END_GET
END_PROPERTY

PROPERTY RunCycle : BOOL
GET
END_GET
SET
END_SET
END_PROPERTY

PROPERTY INTERNAL SafetyOk : BOOL
GET
END_GET
SET
END_SET
END_PROPERTY

PROPERTY StateColor : DWORD
GET
END_GET
END_PROPERTY

PROPERTY PUBLIC Station : E_Station
GET
END_GET
SET
END_SET
END_PROPERTY

PROPERTY Stopped : BOOL
GET
END_GET
END_PROPERTY

PROPERTY TextAuto : ST_Text
GET
END_GET
END_PROPERTY

PROPERTY TextHome : ST_Text
GET
END_GET
END_PROPERTY

PROPERTY PUBLIC TotalCycles : UDINT
GET
END_GET
END_PROPERTY

END_INTERFACE

// ---- POUs/System/Utilities/Interfaces/I_StringBuilder.TcIO
INTERFACE I_StringBuilder

METHOD PUBLIC Append : I_StringBuilder // Append text to the current build string.
VAR_IN_OUT CONSTANT
	text : T_MaxString; // Text to append to current build string
END_VAR
END_METHOD

METHOD PUBLIC AppendAny : I_StringBuilder // Append text to the current build string.
VAR_INPUT
	value : ANY; // Value to append to current build string
END_VAR
END_METHOD

METHOD PUBLIC AppendWs : I_StringBuilder
VAR_IN_OUT CONSTANT
	value : WSTRING;
END_VAR
END_METHOD

METHOD PUBLIC Clear : I_StringBuilder // Clear the current build string.
VAR_INPUT
END_VAR
END_METHOD

METHOD PUBLIC Insert : I_StringBuilder
VAR_INPUT
	text	 : T_MaxString;	// Text to append to current build string
	position : INT;			// Insert position (Index)
END_VAR
END_METHOD

METHOD PUBLIC Reset : I_StringBuilder //Reset current build string to an empty string.
VAR_INPUT
END_VAR
END_METHOD

METHOD PUBLIC Set : I_StringBuilder
VAR_INPUT
	text : T_MaxString; //Text to append to current build string
END_VAR
END_METHOD

METHOD PUBLIC SetWs : I_StringBuilder
VAR_IN_OUT CONSTANT
	value : WSTRING;
END_VAR
END_METHOD

METHOD PUBLIC ToString : T_MaxString // Returns current build string.
VAR_INPUT
END_VAR
END_METHOD

END_INTERFACE

// ---- POUs/System/Utilities/Interfaces/I_WStringBuilder.TcIO
INTERFACE I_WStringBuilder

METHOD PUBLIC Append : I_WStringBuilder // Append text to the current build string.
VAR_INPUT
	text : WSTRING; // Text to append to current build string
END_VAR
END_METHOD

METHOD PUBLIC AppendAny : I_WStringBuilder // Append text to the current build string.
VAR_INPUT
	value : ANY; // Value to append to current build string
END_VAR
END_METHOD

METHOD PUBLIC Clear : I_WStringBuilder // Clear the current build string.
VAR_INPUT
END_VAR
END_METHOD

METHOD PUBLIC Insert : I_WStringBuilder
VAR_INPUT
	text	 : WSTRING;	// Text to append to current build string
	position : INT;		// Insert position (Index)
END_VAR
END_METHOD

METHOD PUBLIC Reset : I_WStringBuilder //Reset current build string to an empty string.
VAR_INPUT
END_VAR
END_METHOD

METHOD PUBLIC Set : I_WStringBuilder
VAR_INPUT
	text : WSTRING; //Text to append to current build string
END_VAR
END_METHOD

METHOD PUBLIC ToString : T_MaxString // Returns current build string.
END_METHOD

METHOD PUBLIC ToWString : WSTRING // Returns current build string.
VAR_INPUT
END_VAR
END_METHOD

END_INTERFACE

// ---- POUs/MAIN.TcPOU
PROGRAM MAIN
VAR	
	/// private var's
	ii						: INT;
	wsClearText				: WSTRING(255);		// clear text for debug
	nOnlineChangesMirror	: UDINT;			// online change tracker
	bInit					: BOOL; 			// PLC init flag
	bRunUnitTest			: BOOL;				// UnitTest
	
	nHmiSize				: ARRAY[0..15] OF UDINT;
END_VAR

///
/// MAIN program - starting point of the PLC project.
/// TP/www.rmth.at/5.2025
/// 

///
/// CHANGES
/// - NAME/DATE/COMMENT

wsClearText := "Run system provider (get time, logger, system and PLC info, ...)";
P_System();

wsClearText := "Init PLC";
M_ChangeWatchdog();

IF NOT M_Init() THEN
	RETURN;
END_IF

wsClearText := "P_Safety";
P_Safety();
	
wsClearText := "Call HMI Controller component";
P_HMI_Controller();

wsClearText := "Call P_Plant";
P_Plant();

wsClearText := "P_Supervision";
P_Supervision(stIO_Cabinet := IO.stControlCabinetIO, nLogger := Services.ILog);

wsClearText := "P_SysSrv";
P_SysSrv();
	
wsClearText := "Run unit tests";
IF bRunUnitTest THEN
	P_UnitTest();
END_IF

Services.b1stShot := FALSE;
Services.bPlcInitDone := TRUE;


(*// DEBUG / TESTS
nHmiSize[0] := SIZEOF(HMI.stHmiInOut);

nHmiSize[1] := SIZEOF(HMI.stHmiTc3);
nHmiSize[2] := SIZEOF(HMI.stHmiTc3.stIn);
nHmiSize[3] := SIZEOF(HMI.stHmiTc3.stOut);

nHmiSize[4] := SIZEOF(HMI.stHmiTc3.stOut.stHeader);
nHmiSize[5] := SIZEOF(HMI.stHmiTc3.stOut.stPopup);
nHmiSize[6] := SIZEOF(HMI.stHmiTc3.stOut.stCounter);
nHmiSize[7] := SIZEOF(HMI.stHmiTc3.stOut.stControlCounter);
nHmiSize[8] := SIZEOF(HMI.stHmiTc3.stOut.stNotificationControl);
nHmiSize[9] := SIZEOF(HMI.stHmiTc3.stOut.stNotificationList);
nHmiSize[10] := SIZEOF(HMI.stHmiTc3.stOut.stNotificationArchiv);
nHmiSize[11] := SIZEOF(HMI.stHmiTc3.stOut.stConditionMonitoring);
nHmiSize[12] := SIZEOF(HMI.stHmiTc3.stOut.stSetupPlant);
nHmiSize[13] := SIZEOF(HMI.stHmiTc3.stOut.stEmergencyStop);
nHmiSize[14] := SIZEOF(HMI.stHmiTc3.stOut.stDoor);
//nHmiSize[15] := SIZEOF(HMI.stHmiTc3.stOut.astStation); *)

ACTION Info:
(*
//----------------------------------------------------------------------

Vorgabe 12.0 s / Stück

Ergebnissdaten Prüflinge: 	iO; Lfd.Nr.;
							
Koordinatensystem Anlage
X = von links nach rechts (Ansicht Vorne)
Y = Vorne (Eingabe) nach hinten
Z = Vertikal						

Stationsauswahl

ST001 Eingabe

----------------------------------------
Schutzbereiche

Schutzbereich 1 -> 	Modul 1 gesamt

//---------------------------------------------------------------------
Anzahl Rund Takt Tisch (RTT) Nestplätze 4 Nester 1

//---------------------------------------------------------------------
Abkürzungen Fehler:
HS = Hochspannung

	
//---------------------------------------------------------------------
pragmas

{text 'todo remove after commissioning'} 
{info 'todo remove after commissioning'} 
{warning 'todo remove after commissioning'} 
{error 'todo remove after commissioning'} 

//----------------------------------------------------------------------

Die wichtigsten Infos zu TC3/RMTH Standard:
	*** min/max und default Werte von Datentypen ***
		RmthTc3Library -> StaticsConstant
		
	*** Stringfunktionen aus RmthTc3Library ***
		aSClearText[EN] := Concat2-10('Text... / ConcatArray(...
		F_RealToString / F_RealToStringEx / F_LRealToString / F_LRealToStringEx
		
	*** Background -> UnitTest ***
		Komponenten hier testen!!!
		
	*** Automatic Sequence Demo ***
		siehe Background -> UnitTest -> TestCases -> StationTest -> FB_TestStation (zb.: DEMO oder M_Sequence)
		
	*** aktuelle PLC System Info ***
		Statics.stPlcSystemInfo
	
--- TC3 Allgemein ---

	*** DATENTYPEN 	***
		https://infosys.beckhoff.com/content/1031/tcplccontrol/html/tcplcctrl_plc_data_types_overview.htm?id=7365416610509907248
	
	*** ATTRIBUTE 	***
		https://infosys.beckhoff.com/content/1031/tc3_plc_intro/54043195664658571.html?id=1095976264130046106
		
	 - Attribut monitoring (Property-OnlineView)
		{attribute 'monitoring' := 'variable'}
		{attribute 'monitoring' := 'call'}
		
		variable: 	Eine implizite Variablen wird angelegt, deren Wert aktualisiert wird, wenn die Applikation die Set oder Get Methode der Eigenschaft aufruft.
		call: 		Der Monitoring-Dienst ruft die Get Methode der Eigenschaft auf
		
		Beispiel:
		{attribute 'monitoring' := 'call'}
		PROPERTY TestState : E_TestCaseState
		
	 - Attribut pack_mode (ändern des Alignments)
		0	aligned, d.h. es treten keine Speicherlücken auf
		1	1-byte-aligned (identisch zu aligned)
		2	2-byte-aligned, d.h. die maximale Größe einer Speicherlücke ist 1 byte
		4	4-byte-aligned, d.h. die maximale Größe einer Speicherlücke ist 3 byte
		8	8-byte-aligned, d.h. die maximale Größe einer Speicherlücke ist 7 byte
		
		Beispiel:
		{attribute 'pack_mode' := '1'}
		TYPE ST_MyStruct:
		
--- Text ---		
		F_CreateDynText("velooffsetchain",0)
		
------------------------------------------------------------------------------------------------------------------------
how to use popup
		
CASE nTestStep OF
	
	0:
		;
	
	10:
		IF fbHmiHandler.M_PopupCheck(E_Popup.ePopup01) THEN
			CASE fbHmiHandler.M_PopupSet(E_Popup.ePopup01,F_CreateDynText("Wasch Prozess Starten ?",0),F_CreateDynText("yes",0),F_CreateDynText("no",0),F_CreateDynText("Info",0),F_CreateDynText("Abbrechen",0)) OF
				1:
					nTestStep :=100;
				2:
					nTestStep :=0;		
				4:	
					nTestStep :=200;
			END_CASE			
		END_IF
	100:
		IF fbHmiHandler.M_PopupCheck(E_Popup.ePopup02) THEN
			CASE fbHmiHandler.M_PopupSet(E_Popup.ePopup02,F_CreateDynText("Wollen Sie wirklich den Wasch Prozess Starten ?? Sicher ??",0),F_CreateDynText("yes",0),F_CreateDynText("",0),F_CreateDynText("Abbruch",0),F_CreateDynText("",0)) OF

				1:
					nTestStep :=200;		
				3:	
					nTestStep :=0;
			END_CASE			
		END_IF
		
	200:
		IF fbHmiHandler.M_PopupCheck(E_Popup.ePopup01) THEN
			CASE fbHmiHandler.M_PopupSet(E_Popup.ePopup01,F_CreateDynText("Prozess Fertig",0),F_CreateDynText("OK",0),F_CreateDynText("",0),F_CreateDynText("",0),F_CreateDynText("",0)) OF
				1:
					nTestStep :=0;
			END_CASE			
		END_IF	
END_CASE

IF FALSE THEN
	IF fbHmiHandler.M_PopupCheck(E_Popup.ePopupSafetyEs) THEN
		fbHmiHandler.M_PopupSet(E_Popup.ePopupSafetyEs,F_CreateDynText("Nothalt nicht OK -> Bitte Quittieren !",0),F_CreateDynText("",0),F_CreateDynText("",0),F_CreateDynText("",0),F_CreateDynText("OK",0)) ;
	END_IF	
END_IF		
		
		
*)
END_ACTION

METHOD PRIVATE M_ChangeWatchdog : BOOL
VAR
END_VAR
wsClearText := "Run onlineChange watchdog";

stPlcAppSystemInfo := Statics.stPlcSystemInfo.stPlcAppSystemInfo;
IF nOnlineChangesMirror <> stPlcAppSystemInfo.OnlineChangeCnt THEN
	wsClearText := "OnlineChange detected -> ReInit!";
	bInit := FALSE;	
	nOnlineChangesMirror := stPlcAppSystemInfo.OnlineChangeCnt;
END_IF
END_METHOD

METHOD PRIVATE M_Init : BOOL
VAR
	// local temp var's
	ISt : IStation;
END_VAR
///
///	PLC INIT: Initialisierung aller Komponenten
/// - Einstellungen treffen
/// - setzen von Referenzen
/// - wichtig: in einem Zyklus fertig!

wsClearText := "Check PLC init done";
IF bInit THEN
	M_Init := TRUE;
	RETURN;
END_IF

wsClearText := "PLC init: first shot setup";
IF Statics.stPlcSystemInfo.stPlcTaskSystemInfo.FirstCycle THEN
	;//P_HMI.recipeManagement.M_ReadRecipe();
END_IF

wsClearText := "PLC init: wait for valid system Time";
IF Statics.dtNow = dtMinValue THEN
	RETURN;
END_IF

{region "configuration and logging"}
wsClearText := "PLC init: setup/load configuration";
stConfig.stLogConfig.eLoggingProvider := E_LoggingProvider.eLoggingProviderFile;
stConfig.stLogConfig.sLogName := 'PlcLog.txt';
stConfig.stLogConfig.sLogPath := '/home/';
stConfig.stLogConfig.eLogLevel := E_LogLevel.eLogLevel_info;

wsClearText := "Set up logging provider";
P_System.fbFileLog.Source := stConfig.stLogConfig.sLogName;
P_System.fbFileLog.sPath := stConfig.stLogConfig.sLogPath;
P_System.fbFileLog.LogLevel := stConfig.stLogConfig.eLogLevel;
	
P_System.fbEventLog.Source := stConfig.stLogConfig.sLogName;
P_System.fbEventLog.LogLevel := stConfig.stLogConfig.eLogLevel;
	
P_System.fbDebugLog.Source := stConfig.stLogConfig.sLogName;
P_System.fbDebugLog.LogLevel := stConfig.stLogConfig.eLogLevel;
IF stConfig.stLogConfig.eLoggingProvider = E_LoggingProvider.eLoggingProviderFile THEN
	Services.ILog := P_System.fbFileLog;
ELSIF stConfig.stLogConfig.eLoggingProvider = E_LoggingProvider.eLoggingProviderEventLog THEN
	Services.ILog := P_System.fbEventLog;
ELSE // default
	Services.ILog := P_System.fbDebugLog;
END_IF

Services.fbEventHandler.Init();

{endregion}

{region "initialize HMI controller and provider"}
wsClearText := "Initialize HMI";
P_HMI_Controller.M_Init();
HMI.fbHmiHwProvider.M_Init();
HMI.fbHmiTc3Provider.M_Init();
{endregion}

{region "initialize components, stations and modules"}

wsClearText := "Initialize plant components";
// plant component initialization here...
	 

wsClearText := "Initialize stations, modules and plant";

// sample 1: quick, default IOs and services:
//		fbSt010OvenA.M_Init();
	 
// sample 2: using custom settings, IOs and services:
//		fbSt010OvenA.Station := E_Station.eStation_ST010_OvenA;
//		fbSt010OvenA.Name := stTextListGlobal.stText_ST010_Name;
//		fbSt010OvenA.Active := TRUE;
//		fbSt010OvenA.Enable := TRUE;
//		fbSt010OvenA.M_SetReferences(IO.st010_OvenA_IO);
//		ISt := fbSt010OvenA.M_InitEx(Services.ILog, Services.fbNotiHandler);
//		fbModul001.M_RegisterStation(ISt);
	 
fbSt010OvenA.M_Init();
fbSt020OvenB.M_Init();
fbSt030Handling.M_Init();
fbSt040Storage.M_Init();
fbSt050Mould.M_Init();
fbModul001.M_Init();
P_Plant.M_Init();

{endregion}

wsClearText := "Initialize Safety";
P_Safety.M_Init();

wsClearText := "Initialize Supervision";
P_Supervision.M_Init();

wsClearText := "PLC init done.";
Services.ILog.AddLog(TO_STRING(wsClearText), sSource, E_LogLevel.eLogLevel_info);

bInit := TRUE;
M_Init := bInit;
END_METHOD

 {attribute 'call_after_online_change_slot' := '1'}
METHOD M_OnlineChange : BOOL
VAR_INPUT
END_VAR
bInit := FALSE;
END_METHOD

END_PROGRAM

// ---- POUs/Safety/P_Safety.TcPOU
PROGRAM P_Safety
VAR_INPUT
	//fbSafetyAccessManager		: ARRAY[1..E_SafetyAccess.eSafetyAccess_nMaxIdx] OF FB_SafetyAccessManager;
	//bDoorRequestSafetyAccess	: ARRAY[1..E_Door.eDoor_nMaxIdx] OF BOOL;
	bDoorOpnS1_3,
	bDoorClsS1_3 				: BOOL;
END_VAR
VAR_OUTPUT
	bError,
	bMachineRequestStart,
	bMachineRequestStop,
	bMachineRequestCycleStop	: BOOL;
	nSchott2StateCol 			: DINT := STATICS.stColor.Gray;
END_VAR
VAR
	/// Safets IOs
	stIO			: REFERENCE TO ST_SafetyIO;

	/// logger & event handler
	ILog			: I_Logger;
	IEvent			: I_EventHandler;
	
	/// private var's
	bSimulation		: BOOL;
	bTestReset		: BOOL;
	aa, ii			: INT;
	nStep			: INT;
	stStepText		: ST_Text;
	
	tofSafetyRun		: ARRAY[0..iSafety_Anzahl_TwinSafeGruppen] OF tof;
	bFBSafeFbErr		: BOOL;
	bFBSafeOutErr		: BOOL;
	bFBSafeComErr		: BOOL;
	bGrpPrtOtherErr		: BOOL;
	
	iResetCnt,
	iErrAckCnt			: INT;
	tonDelay			: TON;	
	
	bEdm_EmergencyStop		: BOOL;
	stEdm_State_Nothalt		: ST_Text;
	arrTonEdmCheck			: ARRAY[0..50] OF TON;
	//arrReleaseDoorOpen	: ARRAY[1..2] OF BOOL; //1=Modul 1 Schott 2= Modul 1 General
	
	fTrigErrorAck			: F_TRIG;
	
	// Safe Gate MBM
	fbSaftyDoors_MGB2		: ARRAY[0..4] OF FB_SafeDoorMGB2;
	fbSaftyDoors			: ARRAY[0..1] OF FB_SafetyDoor;
	
	//fbDoor				: ARRAY[1..E_Door.eDoor_nMaxIdx] OF FB_Door;
	iDoorSequence			: ARRAY[1..iSafety_Anzahl_Schutzbereiche] OF INT;
	tonDoorWait				: ARRAY[1..iSafety_Anzahl_Schutzbereiche] OF TON;
	tonDoorTimeout			: ARRAY[1..iSafety_Anzahl_Schutzbereiche] OF TON;
	
	bTest					: BOOL;
	
	rtrigReset 				: R_TRIG;
	
	tofEsOk,
	tofAreaOkST10,
	tofAreaOkST80 			: TOF;
END_VAR

///
/// HMI access provider
/// 

M_Mapping();

tofEsOk(IN := IO.stSafetyIO.stIn.bSAFE_ES_Ok, PT := T#500MS);
tofAreaOkST10(IN := IO.stSafetyIO.stIn.bSAFE_Area_Ok_ST10, PT := T#2S);

M_Edm();

// run diagnostics
M_Diagnostics();

FOR aa := 1 TO iSafety_Anzahl_Schutzbereiche DO
	tonDoorWait[aa].PT:=T#500MS;
	tonDoorWait[aa]();
	tonDoorWait[aa].IN:=FALSE;
	
	tonDoorTimeout[aa].PT:=T#5000MS;
	tonDoorTimeout[aa]();
	tonDoorTimeout[aa].IN:=FALSE;	
END_FOR


tofSafetyRun[1].IN:=NOT stIO.stOut.bSafetyErrAck[1];
tofSafetyRun[1].PT:=T#4S;
tofSafetyRun[1]();
stIO.stOut.bSafe_Tsg_Run[1]:=tofSafetyRun[1].Q;

// calls
M_DoorSequence();
M_General();

// Simulation ohne HW
IF bSimulation THEN // OR iIBN <> 0 THEN
	stIO.stIn.bSAFE_ES_Ok := TRUE;

	FOR aa := 1 TO iSafety_Anzahl_Schutzbereiche DO
		stIO.stIn.bSAFE_AREA_Ok[aa] := TRUE;
	END_FOR
	
	FOR aa := 1 TO E_Door.eDoor_nMaxIdx DO
		stIO.stIn.bSAFE_GATE_Ok[aa] := TRUE;		
	END_FOR
	
	stIO.stIn.bCompressedAirOk := TRUE;
	

	RETURN; // EXIT
END_IF

// Reset sequence
CASE nStep OF
	0: 	
		stStepText := F_CreateDynText("wait for reset command.", 0);
		IF (HMI.stHmi.stIn.stSafety.bQuitSafety OR bTestReset OR HMI.stHmi.stIn.stMain.stButton_Reset.bClick) THEN
			bTestReset := FALSE;
			bError := FALSE;
			iErrAckCnt := 0;
			nStep := 10;
		END_IF
	
	10:	
		stStepText := F_CreateDynText("Start resetting TwinSAFE", 0);
		IF ErrorAckRequest THEN
			stIO.stOut.bSafetyErrAck[1] := TRUE;			
			nStep := 20;
		ELSE
			nStep := 50;
		END_IF
		
	20:	
		stStepText := F_CreateDynText("Error ack TwinSAFE groups", 0);
		tonDelay(IN := TRUE, PT := T#1S);
		IF tonDelay.Q THEN
			stIO.stOut.bSafetyErrAck[1] := FALSE;
			tonDelay(IN := FALSE);
			IF bFBSafeFbErr OR bFBSafeOutErr OR bFBSafeComErr OR bGrpPrtOtherErr  THEN // chk error still active
				nStep := 30;
			ELSE
				iErrAckCnt := 0;
				nStep := 50;
			END_IF			
		END_IF
		
	30:	
		stStepText := F_CreateDynText("Restart error ack TwinSAFE group", 0);
		tonDelay(IN := TRUE, PT := T#1S);
		IF tonDelay.Q THEN
			tonDelay(IN := FALSE);
			iErrAckCnt := iErrAckCnt + 1;
			IF iErrAckCnt < 3 THEN
				nStep := 10;
			ELSE
				nStep := 0;
			END_IF
		END_IF
		
	50:
		iResetCnt := 0;
		nStep := 55;
		
		
// Restart FBs
		
	55:
		// Feedback NIO
		IF NOT stIO.stIn.bSAFE_ES_Ok AND 
		NOT stIO.stOut.bSafety_EDM_OUT[1] THEN
			IEvent.Select(Tc_Events.TwinSafeEventClass.EdmErrorEvent)
		  	  	  .ArgSbInitWs(stTextListGlobal.stText_Safety.stText_Safety_EDM_Error.wsName)
		  	  	  .ArgSbAppendRaise(' | Safety Feedback Not-Halt');
			nStep := 0;				
		ELSE
			nStep := 56;				
		END_IF

	56:	
		stStepText := F_CreateDynText("Restart TwinSAFE FBs", 0);
		stIO.stOut.bRestartPLC	:= TRUE;
		tonDelay(IN := TRUE, PT := T#0.5S);
		IF tonDelay.Q THEN
			tonDelay(IN := FALSE);
			stIO.stOut.bRestartPLC	:= FALSE;
			nStep := 57;
		END_IF
	57:	
		stStepText := F_CreateDynText("wait", eLanguage);
		tonDelay(IN := TRUE, PT := T#0.2S);
		IF tonDelay.Q THEN
			tonDelay(IN := FALSE);
			IF iResetCnt < 2 THEN // Schleife
				iResetCnt := iResetCnt + 1;
				nStep := 56;
			ELSE			
				nStep := 60;
			END_IF
		END_IF		
		
	60:	
		nStep := 100;
		
	100:
		stStepText := F_CreateDynText("Reset TwinSAFE Done", 0);
		bError := FALSE;
		//stIO.stOut.bMainPressure := TRUE;
		(*// beim ersten Start bestimmte Türen autom. verriegeln wenn geschlossen
		IF NOT bFirstShot THEN
			fbSaftyDoors[2].LockDoor();	// TA Vorne
		END_IF	
		bFirstShot := TRUE;*)
		nStep := 0;
		
END_CASE

{attribute 'monitoring' := 'call'}
PROPERTY INTERNAL CompressedAirOk : BOOL
GET
CompressedAirOk := EmergencyStopOk AND stIO.stIn.bCompressedAirOk;
END_GET
END_PROPERTY

{attribute 'monitoring' := 'call'}
PROPERTY PUBLIC EmergencyStopOk : BOOL
GET // PUBLIC
EmergencyStopOk := tofEsOk.Q;
END_GET
END_PROPERTY

{attribute 'monitoring' := 'call'}
PROPERTY PUBLIC ErrorAckRequest : BOOL
GET
ErrorAckRequest := bFBSafeFbErr OR bFBSafeOutErr OR bFBSafeComErr OR bGrpPrtOtherErr OR 
					NOT stIO.stIn.bSAFE_ES_Ok OR stIO.stIn.bSAFE_DRIVES_STO OR
					stIO.stIn.bSAFE_ConfirmTimeout;
END_GET
END_PROPERTY

METHOD PRIVATE M_Diagnostics : BOOL
VAR_INPUT
END_VAR
// TwinSAFE Fehler										
bFBSafeFbErr :=		IO.stSafetyIO.stIn.bSafe_FbError_Master[0] OR
					IO.stSafetyIO.stIn.bSafe_FbError_Master[1];
					
bFBSafeOutErr :=	IO.stSafetyIO.stIn.bSafe_OutError_Master[0] OR
					IO.stSafetyIO.stIn.bSafe_OutError_Master[1];
					
bFBSafeComErr :=	IO.stSafetyIO.stIn.bSafe_ComError_Master[0] OR
					IO.stSafetyIO.stIn.bSafe_ComError_Master[1];

bGrpPrtOtherErr :=	IO.stSafetyIO.stIn.bSafe_OtherError_Master[0] OR
					IO.stSafetyIO.stIn.bSafe_OtherError_Master[1];
	
// diag ES
IF NOT IO.stSafetyIO.stIn.bSAFE_ES_Ok THEN
	IEvent.Select(Tc_Events.TwinSafeEventClass.ErrorEvent)
		  .ArgSetWString(stTextListGlobal.stText_Safety.stText_Safety_ES.wsName)
		  .Raise();
END_IF

(*	Fehlerauswertung der Sicherheitstechnik

	eNoti_Safety ,
	eNoti_Safety_NotHalt ,
	eNoti_Safety_Schutzbereich ,
	eNoti_Safety_HW ,
	eNoti_Safety_FBs ,
*)
IF stHmi.stIn.stSafety.bQuitSafety THEN
	bError := FALSE;
END_IF

(*	Allgemein - > eNoti_Safety	*)
IF IO.stSafetyIO.stIn.bSafe_EL6900_WcState[0] THEN
	IEvent.Select(Tc_Events.TwinSafeEventClass.HwErrorEvent)
		  .ArgSetString('EL6910 (=A02.K20-1KF1.354) - WC State')
		  .Raise();
	bError := TRUE;

(*	Gruppen FB Fehler	*)
ELSIF IO.stSafetyIO.stIn.bSafe_FbError_Master[0] THEN
	IEvent.Select(Tc_Events.TwinSafeEventClass.ErrorEvent)
		  .ArgSbInitWs(stTextListGlobal.stText_Safety.stText_Safety_Grp_Error.wsName)
		  .ArgSbAppend(' | 000_ES | (=A02.K20-1KF1.354) | ')
		  .ArgSbAppendWsRaise(stTextListGlobal.stText_Safety.stText_Safety_GrpFB_Error.wsName);
	bError := TRUE;
ELSIF IO.stSafetyIO.stIn.bSafe_FbError_Master[1] THEN
	IEvent.Select(Tc_Events.TwinSafeEventClass.ErrorEvent)
		  .ArgSbInitWs(stTextListGlobal.stText_Safety.stText_Safety_Grp_Error.wsName)
		  .ArgSbAppend(' | 000_Areas | (=A02.K20-1KF1.354) | ')
		  .ArgSbAppendWsRaise(stTextListGlobal.stText_Safety.stText_Safety_GrpFB_Error.wsName);
	bError := TRUE;
END_IF


(*	NotHalt Meldungen - > eNoti_Safety_NotHalt	*)
//IF NOT IO.stSafetyIO.stIn.bSafe_EStop_State[E_EmergencyStop.eEmergencyStop_1] THEN
//	IEvent.Select(Tc_Events.TwinSafeEventClass.ErrorEvent)
//		  .ArgSbInitWs(stTextListGlobal.stText_Safety.stText_Safety_ES.wsName)
//		  .ArgSbAppendRaise(' | Schrank | BMK=A01.ES1');
//	bError := TRUE;                                                                             
//ELS

IF NOT IO.stSafetyIO.stIn.bSafe_EStop_State[E_EmergencyStop.eEmergencyStop_2] THEN
	IEvent.Select(Tc_Events.TwinSafeEventClass.ErrorEvent)
		  .ArgSbInitWs(stTextListGlobal.stText_Safety.stText_Safety_ES.wsName)
		  .ArgSbAppendRaise(' | Schrank | BMK=A01.ES2');
	bError := TRUE;
END_IF

// Door/Area Meldungen
IF NOT IO.stSafetyIO.stIn.bSAFE_Area_Ok_ST10 THEN
	IEvent.Select(Tc_Events.TwinSafeEventClass.WarningEvent)
		  .ArgSbInitWs(stTextListGlobal.stText_Safety.stText_Safety_DoorOpen.wsName)
		  .ArgSbAppendRaise(' | Ofen A | BMK=');
END_IF
IF NOT IO.stSafetyIO.stIn.bSAFE_Area_Ok_ST20 THEN
	IEvent.Select(Tc_Events.TwinSafeEventClass.WarningEvent)
		  .ArgSbInitWs(stTextListGlobal.stText_Safety.stText_Safety_DoorOpen.wsName)
		  .ArgSbAppendRaise(' | Ofen B | BMK=');
END_IF

//ToDo: Safety FB's,.. diag
RETURN;

(********	Diagnose Emergency Stop	*********)
fbDiag_NotHalt[1].wsFunctionBlockText := "++A1+P1-6S2 - TSG 000 - ES_Haupt_Pult_1";
fbDiag_NotHalt[2].wsFunctionBlockText := "++M1+P1-2S1 - TSG 000 - ES_Modul_1_Pult_1";
fbDiag_NotHalt[3].wsFunctionBlockText := "++M1+P2-2S1 - TSG 000 - ES_Modul_1_Pult_2";

(********	Diagnose TwoHand	*********)
fbDiag_TwoHand[1].wsFunctionBlockText := "++A1+P1-5S2 - TSG 000 - BA_Tasten - Taste_Betriebsart_Aus";
fbDiag_TwoHand[2].wsFunctionBlockText := "++A1+P1-5S2 - TSG 000 - BA_Tasten - Taste_Betriebsart_Hand";
fbDiag_TwoHand[3].wsFunctionBlockText := "++A1+P1-5S2 - TSG 000 - BA_Tasten - Taste_Betriebsart_Ruest";
fbDiag_TwoHand[4].wsFunctionBlockText := "++A1+P1-5S2 - TSG 000 - BA_Tasten - Taste_Betriebsart_Auto";
fbDiag_TwoHand[5].wsFunctionBlockText := "++A1+P1-6S4 - TSG 000 - BA_Tasten - Taste_P1_Zustimmung_1";
fbDiag_TwoHand[6].wsFunctionBlockText := "++A1+P1-6S6 - TSG 000 - BA_Tasten - Taste_P1_Zustimmung_2";

(********	Diagnose MachineMonitoring	*********)
fbDiag_MachineMonitoring[1].wsFunctionBlockText := "++M1+PSEN_001-2S2 - TSG 000 - Modul1 Tuer 1";
fbDiag_MachineMonitoring[2].wsFunctionBlockText := "++M1+PSEN_002-2S2 - TSG 000 - Modul1 Tuer 2";
fbDiag_MachineMonitoring[3].wsFunctionBlockText := "++M1+PSEN_003-2S2 - TSG 000 - Modul1 Tuer 3";
fbDiag_MachineMonitoring[4].wsFunctionBlockText := "++M1+PSEN_004-2S2 - TSG 000 - Modul1 Tuer 4";
fbDiag_MachineMonitoring[5].wsFunctionBlockText := "++M1+PSEN_005-2S2 - TSG 000 - Modul1 Schott 1";
fbDiag_MachineMonitoring[6].wsFunctionBlockText := "++M1+E2-73BG7 - TSG 000 - Modul1 Schott 2";


(********	Diagnose EDM	*********)
//fbDiag_EDM[1].wsFunctionBlockText := ""; // Not-Halt = wird über ES Baustein überwacht
fbDiag_EDM[1].wsFunctionBlockText := "++M1+E1-80K3K4 - TSG 002 - Edm Pilotluft Lastspannung_Modul 1";
fbDiag_EDM[2].wsFunctionBlockText := "++M1+E1-80K3K4 - TSG 002 - Edm Rtt";

(*	Logik	*)

(*	FB Details	*)
(*	Autoquitt		*)
FOR aa := 1 TO iSafetyDiag_Anzahl_FbEmergencyStop DO

	(*	Not-Halt Diagnose		*)
	fbDiag_NotHalt[aa].stIn := Iarr_SafetyDiag_NotHalt[aa];
	fbDiag_NotHalt[aa]( );
	(*	Error anzeigen	*)
	IF fbDiag_NotHalt[aa].bError THEN
		IEvent.Select(Tc_Events.TwinSafeEventClass.ErrorEvent)
			  .ArgSbInitWs(stTextListGlobal.stText_Safety.stText_Safety_FB_Error.wsName)
		  	  .ArgSbAppend(' | ')
			  .ArgSbAppendWsRaise(fbDiag_NotHalt[aa].stErrorText.wsName);
	END_IF
END_FOR

FOR aa := 0 TO iSafetyDiag_Anzahl_FbMachineMonitoring DO
	(*	MachineMonitoring (Schutztürbaustein) Diagnose		*)
	fbDiag_MachineMonitoring[aa].stIn := Iarr_SafetyDiag_MachineMonitoring[aa];
	fbDiag_MachineMonitoring[aa]( );
	(*	Error anzeigen	*)
	IF fbDiag_MachineMonitoring[aa].bError THEN
		IEvent.Select(Tc_Events.TwinSafeEventClass.ErrorEvent)
			  .ArgSbInitWs(stTextListGlobal.stText_Safety.stText_Safety_FB_Error.wsName)
		  	  .ArgSbAppend(' | ')
			  .ArgSbAppendWsRaise(fbDiag_MachineMonitoring[aa].stErrorText.wsName);
	END_IF
END_FOR

